LIN {X 0,Y 310.655,Z 525.848,A -85,B 0,C 180,E1 -15761.749,E2 -15761.749} C_VEL
LIN {X 0,Y 310.622,Z 526.997,A -85,B 0,C 180,E1 -15763.368,E2 -15763.368} C_VEL
LIN {X 0,Y 310.6,Z 527.515,A -85,B 0,C 180,E1 -15765.756,E2 -15765.756} C_VEL
LIN {X 0,Y 310.891,Z 526.626,A -85,B 0,C 180,E1 -15768.294,E2 -15768.294} C_VEL
LIN {X 0,Y 311.191,Z 525.391,A -85,B 0,C 180,E1 -15769.802,E2 -15769.802} C_VEL
LIN {X 0,Y 311.807,Z 522.832,A -85,B 0,C 180,E1 -15771.834,E2 -15771.834} C_VEL
LIN {X 0,Y 312.562,Z 519.175,A -85,B 0,C 180,E1 -15773.875,E2 -15773.875} C_VEL
LIN {X 0,Y 313.548,Z 514.547,A -85,B 0,C 180,E1 -15775.824,E2 -15775.824} C_VEL
LIN {X 0,Y 314.939,Z 508.045,A -85,B 0,C 180,E1 -15777.946,E2 -15777.946} C_VEL
LIN {X 0,Y 316.348,Z 501.394,A -85,B 0,C 180,E1 -15779.675,E2 -15779.675} C_VEL
LIN {X 0,Y 317.833,Z 493.733,A -85,B 0,C 180,E1 -15781.308,E2 -15781.308} C_VEL
LIN {X 0,Y 319.671,Z 484.109,A -85,B 0,C 180,E1 -15782.966,E2 -15782.966} C_VEL
LIN {X 0,Y 321.573,Z 473.195,A -85,B 0,C 180,E1 -15784.445,E2 -15784.445} C_VEL
LIN {X 0,Y 323.064,Z 462.681,A -85,B 0,C 180,E1 -15785.587,E2 -15785.587} C_VEL
LIN {X 0,Y 324.486,Z 450.756,A -85,B 0,C 180,E1 -15786.597,E2 -15786.597} C_VEL
LIN {X 0,Y 325.603,Z 438.12,A -85,B 0,C 180,E1 -15787.378,E2 -15787.378} C_VEL
LIN {X 0,Y 326.342,Z 425.507,A -85,B 0,C 180,E1 -15787.912,E2 -15787.912} C_VEL
LIN {X 0,Y 327.507,Z 389.604,A -85,B 0,C 180,E1 -15788.742,E2 -15788.742} C_VEL
LIN {X 0,Y 328.624,Z 348.659,A -85,B 0,C 180,E1 -15789.655,E2 -15789.655} C_VEL
LIN {X 0,Y 322.438,Z 334.155,A -85,B 0,C 180,E1 -15790.674,E2 -15790.674} C_VEL
LIN {X 0,Y 315.363,Z 320.101,A -85,B 0,C 180,E1 -15791.839,E2 -15791.839} C_VEL
LIN {X 0,Y 314.876,Z 319.253,A -85,B 0,C 180,E1 -15791.919,E2 -15791.919} C_VEL
LIN {X 0,Y 313.157,Z 317.364,A -85,B 0,C 180,E1 -15792.239,E2 -15792.239} C_VEL
LIN {X 0,Y 310.38,Z 316.136,A -85,B 0,C 180,E1 -15792.856,E2 -15792.856} C_VEL
LIN {X 0,Y 306.923,Z 314.284,A -85,B 0,C 180,E1 -15793.938,E2 -15793.938} C_VEL
LIN {X 0,Y 305.535,Z 312.708,A -85,B 0,C 180,E1 -15794.807,E2 -15794.807} C_VEL
LIN {X 0,Y 305.384,Z 312.449,A -85,B 0,C 180,E1 -15795.209,E2 -15795.209} C_VEL
LIN {X 0,Y 305.443,Z 312.442,A -85,B 0,C 180,E1 -15798.143,E2 -15798.143} C_VEL
LIN {X 0,Y 305.478,Z 312.425,A -85,B 0,C 180,E1 -15801.598,E2 -15801.598} C_VEL
LIN {X 0,Y 305.464,Z 312.435,A -85,B 0,C 180,E1 -15804.887,E2 -15804.887} C_VEL
LIN {X 0,Y 305.454,Z 312.436,A -85,B 0,C 180,E1 -15808.355,E2 -15808.355} C_VEL
LIN {X 0,Y 305.523,Z 312.427,A -85,B 0,C 180,E1 -15811.114,E2 -15811.114} C_VEL
LIN {X 0,Y 305.573,Z 312.418,A -85,B 0,C 180,E1 -15814.088,E2 -15814.088} C_VEL
LIN {X 0,Y 305.502,Z 312.427,A -85,B 0,C 180,E1 -15818.403,E2 -15818.403} C_VEL
LIN {X 0,Y 305.592,Z 312.409,A -85,B 0,C 180,E1 -15821.218,E2 -15821.218} C_VEL
LIN {X 0,Y 305.65,Z 312.401,A -85,B 0,C 180,E1 -15825.349,E2 -15825.349} C_VEL
LIN {X 0,Y 305.64,Z 312.406,A -85,B 0,C 180,E1 -15829.4,E2 -15829.4} C_VEL
LIN {X 0,Y 305.815,Z 312.388,A -85,B 0,C 180,E1 -15832.074,E2 -15832.074} C_VEL
LIN {X 0,Y 305.688,Z 312.4,A -85,B 0,C 180,E1 -15834.723,E2 -15834.723} C_VEL
LIN {X 0,Y 305.956,Z 312.37,A -85,B 0,C 180,E1 -15838.684,E2 -15838.684} C_VEL
LIN {X 0,Y 305.956,Z 312.357,A -85,B 0,C 180,E1 -15841.316,E2 -15841.316} C_VEL
LIN {X 0,Y 305.852,Z 312.373,A -85,B 0,C 180,E1 -15846.597,E2 -15846.597} C_VEL
LIN {X 0,Y 305.737,Z 312.396,A -85,B 0,C 180,E1 -15849.26,E2 -15849.26} C_VEL
LIN {X 0,Y 305.59,Z 312.416,A -85,B 0,C 180,E1 -15853.296,E2 -15853.296} C_VEL
LIN {X 0,Y 305.595,Z 312.407,A -85,B 0,C 180,E1 -15856.02,E2 -15856.02} C_VEL
LIN {X 0,Y 305.577,Z 312.418,A -85,B 0,C 180,E1 -15859.444,E2 -15859.444} C_VEL
LIN {X 0,Y 305.488,Z 312.434,A -85,B 0,C 180,E1 -15863.039,E2 -15863.039} C_VEL
LIN {X 0,Y 305.528,Z 312.416,A -85,B 0,C 180,E1 -15866.219,E2 -15866.219} C_VEL
LIN {X 0,Y 305.497,Z 312.424,A -85,B 0,C 180,E1 -15869.05,E2 -15869.05} C_VEL
LIN {X 0,Y 305.446,Z 312.436,A -85,B 0,C 180,E1 -15871.952,E2 -15871.952} C_VEL
LIN {X 0,Y 305.464,Z 312.432,A -85,B 0,C 180,E1 -15875.113,E2 -15875.113} C_VEL
LIN {X 0,Y 305.45,Z 312.435,A -85,B 0,C 180,E1 -15878.528,E2 -15878.528} C_VEL
LIN {X 0,Y 305.457,Z 312.437,A -85,B 0,C 180,E1 -15882.586,E2 -15882.586} C_VEL
LIN {X 0,Y 305.427,Z 312.438,A -85,B 0,C 180,E1 -15886.345,E2 -15886.345} C_VEL
LIN {X 0,Y 305.46,Z 312.429,A -85,B 0,C 180,E1 -15889.892,E2 -15889.892} C_VEL
LIN {X 0,Y 305.499,Z 312.616,A -85,B 0,C 180,E1 -15893.627,E2 -15893.627} C_VEL
LIN {X 0,Y 308.251,Z 323.052,A -85,B 0,C 180,E1 -15897.288,E2 -15897.288} C_VEL
LIN {X 0,Y 310.521,Z 332.941,A -85,B 0,C 180,E1 -15900.51,E2 -15900.51} C_VEL
LIN {X 0,Y 311.361,Z 336.906,A -85,B 0,C 180,E1 -15901.679,E2 -15901.679} C_VEL
LIN {X 0,Y 314.684,Z 344.996,A -85,B 0,C 180,E1 -15902.285,E2 -15902.285} C_VEL
LIN {X 0,Y 319.531,Z 367.922,A -85,B 0,C 180,E1 -15903.422,E2 -15903.422} C_VEL
LIN {X 0,Y 321.715,Z 382.032,A -85,B 0,C 180,E1 -15904.015,E2 -15904.015} C_VEL
LIN {X 0,Y 319.792,Z 445.993,A -85,B 0,C 180,E1 -15905.492,E2 -15905.492} C_VEL
LIN {X 0,Y 318.71,Z 459.732,A -85,B 0,C 180,E1 -15906.053,E2 -15906.053} C_VEL
LIN {X 0,Y 317.279,Z 472.616,A -85,B 0,C 180,E1 -15906.847,E2 -15906.847} C_VEL
LIN {X 0,Y 315.482,Z 485.127,A -85,B 0,C 180,E1 -15907.918,E2 -15907.918} C_VEL
LIN {X 0,Y 313.614,Z 496.298,A -85,B 0,C 180,E1 -15909.16,E2 -15909.16} C_VEL
LIN {X 0,Y 311.639,Z 506.4,A -85,B 0,C 180,E1 -15910.57,E2 -15910.57} C_VEL
LIN {X 0,Y 309.74,Z 515.84,A -85,B 0,C 180,E1 -15912.23,E2 -15912.23} C_VEL
LIN {X 0,Y 308.099,Z 524.424,A -85,B 0,C 180,E1 -15914.113,E2 -15914.113} C_VEL
LIN {X 0,Y 306.566,Z 531.627,A -85,B 0,C 180,E1 -15916.071,E2 -15916.071} C_VEL
LIN {X 0,Y 305.309,Z 537.408,A -85,B 0,C 180,E1 -15918.042,E2 -15918.042} C_VEL
LIN {X 0,Y 304.501,Z 541.984,A -85,B 0,C 180,E1 -15920.031,E2 -15920.031} C_VEL
LIN {X 0,Y 303.991,Z 545.486,A -85,B 0,C 180,E1 -15922.026,E2 -15922.026} C_VEL
LIN {X 0,Y 303.66,Z 548.358,A -85,B 0,C 180,E1 -15924.388,E2 -15924.388} C_VEL
LIN {X 0,Y 303.633,Z 549.588,A -85,B 0,C 180,E1 -15926.017,E2 -15926.017} C_VEL
LIN {X 0,Y 303.623,Z 550.172,A -85,B 0,C 180,E1 -15927.346,E2 -15927.346} C_VEL
LIN {X 0,Y 303.607,Z 550.326,A -85,B 0,C 180,E1 -15928.673,E2 -15928.673} C_VEL
LIN {X 0,Y 303.669,Z 550.081,A -85,B 0,C 180,E1 -15929.999,E2 -15929.999} C_VEL
LIN {X 0,Y 303.635,Z 549.443,A -85,B 0,C 180,E1 -15931.325,E2 -15931.325} C_VEL
LIN {X 0,Y 303.645,Z 548.412,A -85,B 0,C 180,E1 -15932.652,E2 -15932.652} C_VEL
LIN {X 0,Y 303.67,Z 546.932,A -85,B 0,C 180,E1 -15933.98,E2 -15933.98} C_VEL
LIN {X 0,Y 303.729,Z 544.305,A -85,B 0,C 180,E1 -15935.743,E2 -15935.743} C_VEL
LIN {X 0,Y 303.938,Z 539.781,A -85,B 0,C 180,E1 -15937.974,E2 -15937.974} C_VEL
LIN {X 0,Y 304.438,Z 533.452,A -85,B 0,C 180,E1 -15940.305,E2 -15940.305} C_VEL
LIN {X 0,Y 305.125,Z 526.543,A -85,B 0,C 180,E1 -15942.3,E2 -15942.3} C_VEL
LIN {X 0,Y 306.006,Z 519.49,A -85,B 0,C 180,E1 -15943.953,E2 -15943.953} C_VEL
LIN {X 0,Y 307.069,Z 510.98,A -85,B 0,C 180,E1 -15945.599,E2 -15945.599} C_VEL
LIN {X 0,Y 308.256,Z 500.429,A -85,B 0,C 180,E1 -15947.24,E2 -15947.24} C_VEL
LIN {X 0,Y 309.191,Z 491.41,A -85,B 0,C 180,E1 -15948.383,E2 -15948.383} C_VEL
LIN {X 0,Y 310.442,Z 480.31,A -85,B 0,C 180,E1 -15949.506,E2 -15949.506} C_VEL
LIN {X 0,Y 311.569,Z 467.989,A -85,B 0,C 180,E1 -15950.463,E2 -15950.463} C_VEL
LIN {X 0,Y 312.495,Z 455.009,A -85,B 0,C 180,E1 -15951.175,E2 -15951.175} C_VEL
LIN {X 0,Y 313.083,Z 441.167,A -85,B 0,C 180,E1 -15951.652,E2 -15951.652} C_VEL
LIN {X 0,Y 314.281,Z 378.975,A -85,B 0,C 180,E1 -15953.068,E2 -15953.068} C_VEL
LIN {X 0,Y 308.693,Z 337.549,A -85,B 0,C 180,E1 -15954.448,E2 -15954.448} C_VEL
LIN {X 0,Y 309.29,Z 331.837,A -85,B 0,C 180,E1 -15955.938,E2 -15955.938} C_VEL
LIN {X 0,Y 307.581,Z 322.176,A -85,B 0,C 180,E1 -15958.673,E2 -15958.673} C_VEL
LIN {X 0,Y 305.465,Z 312.437,A -85,B 0,C 180,E1 -15961.578,E2 -15961.578} C_VEL
LIN {X 0,Y 305.459,Z 312.433,A -85,B 0,C 180,E1 -15965.112,E2 -15965.112} C_VEL
LIN {X 0,Y 305.463,Z 312.435,A -85,B 0,C 180,E1 -15968.532,E2 -15968.532} C_VEL
LIN {X 0,Y 305.45,Z 312.438,A -85,B 0,C 180,E1 -15972.585,E2 -15972.585} C_VEL
LIN {X 0,Y 305.468,Z 312.432,A -85,B 0,C 180,E1 -15977.409,E2 -15977.409} C_VEL
LIN {X 0,Y 305.489,Z 312.428,A -85,B 0,C 180,E1 -15981.599,E2 -15981.599} C_VEL
LIN {X 0,Y 305.457,Z 312.437,A -85,B 0,C 180,E1 -15984.886,E2 -15984.886} C_VEL
LIN {X 0,Y 305.449,Z 312.434,A -85,B 0,C 180,E1 -15988.353,E2 -15988.353} C_VEL
LIN {X 0,Y 305.514,Z 312.429,A -85,B 0,C 180,E1 -15991.113,E2 -15991.113} C_VEL
LIN {X 0,Y 305.564,Z 312.419,A -85,B 0,C 180,E1 -15994.087,E2 -15994.087} C_VEL
LIN {X 0,Y 305.492,Z 312.429,A -85,B 0,C 180,E1 -15998.402,E2 -15998.402} C_VEL
LIN {X 0,Y 305.582,Z 312.418,A -85,B 0,C 180,E1 -16001.217,E2 -16001.217} C_VEL
LIN {X 0,Y 305.641,Z 312.413,A -85,B 0,C 180,E1 -16005.349,E2 -16005.349} C_VEL
LIN {X 0,Y 305.63,Z 312.416,A -85,B 0,C 180,E1 -16009.399,E2 -16009.399} C_VEL
LIN {X 0,Y 305.804,Z 312.386,A -85,B 0,C 180,E1 -16012.074,E2 -16012.074} C_VEL
LIN {X 0,Y 305.68,Z 312.399,A -85,B 0,C 180,E1 -16014.723,E2 -16014.723} C_VEL
LIN {X 0,Y 305.948,Z 312.371,A -85,B 0,C 180,E1 -16018.684,E2 -16018.684} C_VEL
LIN {X 0,Y 305.949,Z 312.373,A -85,B 0,C 180,E1 -16021.316,E2 -16021.316} C_VEL
LIN {X 0,Y 305.666,Z 312.402,A -85,B 0,C 180,E1 -16025.277,E2 -16025.277} C_VEL
LIN {X 0,Y 305.755,Z 312.396,A -85,B 0,C 180,E1 -16027.927,E2 -16027.927} C_VEL
LIN {X 0,Y 305.595,Z 312.42,A -85,B 0,C 180,E1 -16031.946,E2 -16031.946} C_VEL
LIN {X 0,Y 305.63,Z 312.409,A -85,B 0,C 180,E1 -16035.035,E2 -16035.035} C_VEL
LIN {X 0,Y 305.568,Z 312.419,A -85,B 0,C 180,E1 -16039.445,E2 -16039.445} C_VEL
LIN {X 0,Y 305.479,Z 312.43,A -85,B 0,C 180,E1 -16043.04,E2 -16043.04} C_VEL
LIN {X 0,Y 305.54,Z 312.427,A -85,B 0,C 180,E1 -16046.228,E2 -16046.228} C_VEL
LIN {X 0,Y 305.489,Z 312.429,A -85,B 0,C 180,E1 -16049.051,E2 -16049.051} C_VEL
LIN {X 0,Y 305.458,Z 312.43,A -85,B 0,C 180,E1 -16053.518,E2 -16053.518} C_VEL
LIN {X 0,Y 305.463,Z 312.436,A -85,B 0,C 180,E1 -16056.741,E2 -16056.741} C_VEL
LIN {X 0,Y 305.403,Z 312.442,A -85,B 0,C 180,E1 -16060.591,E2 -16060.591} C_VEL
LIN {X 0,Y 305.416,Z 312.436,A -85,B 0,C 180,E1 -16063.657,E2 -16063.657} C_VEL
LIN {X 0,Y 305.431,Z 312.437,A -85,B 0,C 180,E1 -16067.42,E2 -16067.42} C_VEL
LIN {X 0,Y 305.456,Z 312.434,A -85,B 0,C 180,E1 -16071.596,E2 -16071.596} C_VEL
LIN {X 0,Y 305.459,Z 312.436,A -85,B 0,C 180,E1 -16074.888,E2 -16074.888} C_VEL
LIN {X 0,Y 305.439,Z 312.435,A -85,B 0,C 180,E1 -16078.36,E2 -16078.36} C_VEL
LIN {X 0,Y 305.472,Z 312.434,A -85,B 0,C 180,E1 -16081.11,E2 -16081.11} C_VEL
LIN {X 0,Y 305.496,Z 312.429,A -85,B 0,C 180,E1 -16084.083,E2 -16084.083} C_VEL
LIN {X 0,Y 305.472,Z 312.433,A -85,B 0,C 180,E1 -16086.977,E2 -16086.977} C_VEL
LIN {X 0,Y 305.542,Z 312.425,A -85,B 0,C 180,E1 -16091.216,E2 -16091.216} C_VEL
LIN {X 0,Y 305.628,Z 312.415,A -85,B 0,C 180,E1 -16095.349,E2 -16095.349} C_VEL
LIN {X 0,Y 305.627,Z 312.566,A -85,B 0,C 180,E1 -16098.225,E2 -16098.225} C_VEL
LIN {X 0,Y 306.516,Z 316.718,A -85,B 0,C 180,E1 -16099.508,E2 -16099.508} C_VEL
LIN {X 0,Y 312.875,Z 335.486,A -85,B 0,C 180,E1 -16100.394,E2 -16100.394} C_VEL
LIN {X 0,Y 314.978,Z 347.517,A -85,B 0,C 180,E1 -16100.819,E2 -16100.819} C_VEL
LIN {X 0,Y 313.14,Z 424.528,A -85,B 0,C 180,E1 -16102.586,E2 -16102.586} C_VEL
LIN {X 0,Y 312.537,Z 437.514,A -85,B 0,C 180,E1 -16103.14,E2 -16103.14} C_VEL
LIN {X 0,Y 311.726,Z 450.087,A -85,B 0,C 180,E1 -16103.935,E2 -16103.935} C_VEL
LIN {X 0,Y 310.797,Z 461.998,A -85,B 0,C 180,E1 -16104.968,E2 -16104.968} C_VEL
LIN {X 0,Y 309.618,Z 473.529,A -85,B 0,C 180,E1 -16106.259,E2 -16106.259} C_VEL
LIN {X 0,Y 308.386,Z 483.881,A -85,B 0,C 180,E1 -16107.715,E2 -16107.715} C_VEL
LIN {X 0,Y 307.181,Z 493.179,A -85,B 0,C 180,E1 -16109.346,E2 -16109.346} C_VEL
LIN {X 0,Y 306.032,Z 502.185,A -85,B 0,C 180,E1 -16111.317,E2 -16111.317} C_VEL
LIN {X 0,Y 305.201,Z 509.434,A -85,B 0,C 180,E1 -16113.301,E2 -16113.301} C_VEL
LIN {X 0,Y 304.55,Z 515.23,A -85,B 0,C 180,E1 -16115.297,E2 -16115.297} C_VEL
LIN {X 0,Y 304.145,Z 519.658,A -85,B 0,C 180,E1 -16117.236,E2 -16117.236} C_VEL
LIN {X 0,Y 303.766,Z 523.266,A -85,B 0,C 180,E1 -16119.321,E2 -16119.321} C_VEL
LIN {X 0,Y 303.584,Z 524.997,A -85,B 0,C 180,E1 -16120.674,E2 -16120.674} C_VEL
LIN {X 0,Y 303.542,Z 526.313,A -85,B 0,C 180,E1 -16122.028,E2 -16122.028} C_VEL
LIN {X 0,Y 303.531,Z 527.273,A -85,B 0,C 180,E1 -16123.473,E2 -16123.473} C_VEL
LIN {X 0,Y 303.531,Z 527.757,A -85,B 0,C 180,E1 -16126.133,E2 -16126.133} C_VEL
LIN {X 0,Y 303.866,Z 526.883,A -85,B 0,C 180,E1 -16128.508,E2 -16128.508} C_VEL
LIN {X 0,Y 304.21,Z 525.403,A -85,B 0,C 180,E1 -16130.276,E2 -16130.276} C_VEL
LIN {X 0,Y 305.079,Z 521.93,A -85,B 0,C 180,E1 -16132.858,E2 -16132.858} C_VEL
LIN {X 0,Y 306.084,Z 517.421,A -85,B 0,C 180,E1 -16135.137,E2 -16135.137} C_VEL
LIN {X 0,Y 307.33,Z 511.945,A -85,B 0,C 180,E1 -16137.217,E2 -16137.217} C_VEL
LIN {X 0,Y 308.942,Z 504.997,A -85,B 0,C 180,E1 -16139.282,E2 -16139.282} C_VEL
LIN {X 0,Y 310.561,Z 497.418,A -85,B 0,C 180,E1 -16141.088,E2 -16141.088} C_VEL
LIN {X 0,Y 312.218,Z 489.107,A -85,B 0,C 180,E1 -16142.7,E2 -16142.7} C_VEL
LIN {X 0,Y 314.216,Z 478.662,A -85,B 0,C 180,E1 -16144.313,E2 -16144.313} C_VEL
LIN {X 0,Y 316.11,Z 467.254,A -85,B 0,C 180,E1 -16145.705,E2 -16145.705} C_VEL
LIN {X 0,Y 317.626,Z 455.882,A -85,B 0,C 180,E1 -16146.793,E2 -16146.793} C_VEL
LIN {X 0,Y 318.875,Z 444.501,A -85,B 0,C 180,E1 -16147.615,E2 -16147.615} C_VEL
LIN {X 0,Y 319.822,Z 431.965,A -85,B 0,C 180,E1 -16148.274,E2 -16148.274} C_VEL
LIN {X 0,Y 320.387,Z 419.421,A -85,B 0,C 180,E1 -16148.696,E2 -16148.696} C_VEL
LIN {X 0,Y 322.479,Z 350.403,A -85,B 0,C 180,E1 -16150.251,E2 -16150.251} C_VEL
LIN {X 0,Y 315.024,Z 333.6,A -85,B 0,C 180,E1 -16151.517,E2 -16151.517} C_VEL
LIN {X 0,Y 308.345,Z 320.625,A -85,B 0,C 180,E1 -16152.669,E2 -16152.669} C_VEL
LIN {X 0,Y 306.666,Z 317.222,A -85,B 0,C 180,E1 -16153.018,E2 -16153.018} C_VEL
LIN {X 0,Y 305.38,Z 312.451,A -85,B 0,C 180,E1 -16154.77,E2 -16154.77} C_VEL
LIN {X 0,Y 305.384,Z 312.449,A -85,B 0,C 180,E1 -16155.209,E2 -16155.209} C_VEL
LIN {X 0,Y 304.768,Z 312.52,A -85,B 0,C 180,E1 -16156.31,E2 -16156.31} C_VEL
LIN {X 0,Y 301.968,Z 312.875,A -85,B 0,C 180,E1 -16158.104,E2 -16158.104} C_VEL
LIN {X 0,Y 299.556,Z 313.166,A -85,B 0,C 180,E1 -16159.559,E2 -16159.559} C_VEL
LIN {X 0,Y 298.499,Z 313.29,A -85,B 0,C 180,E1 -16160.686,E2 -16160.686} C_VEL
LIN {X 0,Y 298.403,Z 313.302,A -85,B 0,C 180,E1 -16161.068,E2 -16161.068} C_VEL
LIN {X 0,Y 298.421,Z 313.311,A -85,B 0,C 180,E1 -16163.93,E2 -16163.93} C_VEL
LIN {X 0,Y 298.398,Z 313.315,A -85,B 0,C 180,E1 -16167.983,E2 -16167.983} C_VEL
LIN {X 0,Y 298.466,Z 313.306,A -85,B 0,C 180,E1 -16171.904,E2 -16171.904} C_VEL
LIN {X 0,Y 298.488,Z 313.304,A -85,B 0,C 180,E1 -16174.924,E2 -16174.924} C_VEL
LIN {X 0,Y 298.452,Z 313.308,A -85,B 0,C 180,E1 -16179.315,E2 -16179.315} C_VEL
LIN {X 0,Y 298.54,Z 313.293,A -85,B 0,C 180,E1 -16182.179,E2 -16182.179} C_VEL
LIN {X 0,Y 298.595,Z 313.282,A -85,B 0,C 180,E1 -16184.995,E2 -16184.995} C_VEL
LIN {X 0,Y 298.595,Z 313.287,A -85,B 0,C 180,E1 -16189.147,E2 -16189.147} C_VEL
LIN {X 0,Y 298.761,Z 313.264,A -85,B 0,C 180,E1 -16191.886,E2 -16191.886} C_VEL
LIN {X 0,Y 298.66,Z 313.275,A -85,B 0,C 180,E1 -16194.599,E2 -16194.599} C_VEL
LIN {X 0,Y 298.923,Z 313.247,A -85,B 0,C 180,E1 -16198.653,E2 -16198.653} C_VEL
LIN {X 0,Y 298.923,Z 313.233,A -85,B 0,C 180,E1 -16201.347,E2 -16201.347} C_VEL
LIN {X 0,Y 298.798,Z 313.252,A -85,B 0,C 180,E1 -16206.754,E2 -16206.754} C_VEL
LIN {X 0,Y 298.682,Z 313.275,A -85,B 0,C 180,E1 -16209.48,E2 -16209.48} C_VEL
LIN {X 0,Y 298.553,Z 313.292,A -85,B 0,C 180,E1 -16213.615,E2 -16213.615} C_VEL
LIN {X 0,Y 298.55,Z 313.284,A -85,B 0,C 180,E1 -16216.409,E2 -16216.409} C_VEL
LIN {X 0,Y 298.512,Z 313.298,A -85,B 0,C 180,E1 -16219.654,E2 -16219.654} C_VEL
LIN {X 0,Y 298.43,Z 313.31,A -85,B 0,C 180,E1 -16223.6,E2 -16223.6} C_VEL
LIN {X 0,Y 298.487,Z 313.295,A -85,B 0,C 180,E1 -16226.575,E2 -16226.575} C_VEL
LIN {X 0,Y 298.422,Z 313.301,A -85,B 0,C 180,E1 -16229.641,E2 -16229.641} C_VEL
LIN {X 0,Y 298.397,Z 313.312,A -85,B 0,C 180,E1 -16232.8,E2 -16232.8} C_VEL
LIN {X 0,Y 298.448,Z 313.305,A -85,B 0,C 180,E1 -16236.807,E2 -16236.807} C_VEL
LIN {X 0,Y 298.389,Z 313.313,A -85,B 0,C 180,E1 -16241.087,E2 -16241.087} C_VEL
LIN {X 0,Y 298.401,Z 313.313,A -85,B 0,C 180,E1 -16243.103,E2 -16243.103} C_VEL
LIN {X 0,Y 298.405,Z 313.315,A -85,B 0,C 180,E1 -16246.921,E2 -16246.921} C_VEL
LIN {X 0,Y 298.401,Z 313.303,A -85,B 0,C 180,E1 -16251.007,E2 -16251.007} C_VEL
LIN {X 0,Y 298.415,Z 313.327,A -85,B 0,C 180,E1 -16252.777,E2 -16252.777} C_VEL
LIN {X 0,Y 300.934,Z 322.839,A -85,B 0,C 180,E1 -16256.252,E2 -16256.252} C_VEL
LIN {X 0,Y 303.379,Z 333.131,A -85,B 0,C 180,E1 -16259.744,E2 -16259.744} C_VEL
LIN {X 0,Y 304.133,Z 336.54,A -85,B 0,C 180,E1 -16260.785,E2 -16260.785} C_VEL
LIN {X 0,Y 308.933,Z 347.604,A -85,B 0,C 180,E1 -16261.683,E2 -16261.683} C_VEL
LIN {X 0,Y 313.606,Z 370.116,A -85,B 0,C 180,E1 -16262.833,E2 -16262.833} C_VEL
LIN {X 0,Y 315.577,Z 383.159,A -85,B 0,C 180,E1 -16263.394,E2 -16263.394} C_VEL
LIN {X 0,Y 313.642,Z 445.184,A -85,B 0,C 180,E1 -16264.846,E2 -16264.846} C_VEL
LIN {X 0,Y 312.571,Z 458.354,A -85,B 0,C 180,E1 -16265.375,E2 -16265.375} C_VEL
LIN {X 0,Y 311.074,Z 471.572,A -85,B 0,C 180,E1 -16266.181,E2 -16266.181} C_VEL
LIN {X 0,Y 309.419,Z 482.714,A -85,B 0,C 180,E1 -16267.109,E2 -16267.109} C_VEL
LIN {X 0,Y 307.49,Z 494.272,A -85,B 0,C 180,E1 -16268.373,E2 -16268.373} C_VEL
LIN {X 0,Y 305.394,Z 504.704,A -85,B 0,C 180,E1 -16269.806,E2 -16269.806} C_VEL
LIN {X 0,Y 303.365,Z 514.296,A -85,B 0,C 180,E1 -16271.459,E2 -16271.459} C_VEL
LIN {X 0,Y 301.744,Z 522.177,A -85,B 0,C 180,E1 -16273.151,E2 -16273.151} C_VEL
LIN {X 0,Y 300.184,Z 529.466,A -85,B 0,C 180,E1 -16275.075,E2 -16275.075} C_VEL
LIN {X 0,Y 298.735,Z 535.606,A -85,B 0,C 180,E1 -16277.085,E2 -16277.085} C_VEL
LIN {X 0,Y 297.743,Z 540.503,A -85,B 0,C 180,E1 -16279.114,E2 -16279.114} C_VEL
LIN {X 0,Y 297.09,Z 544.302,A -85,B 0,C 180,E1 -16281.154,E2 -16281.154} C_VEL
LIN {X 0,Y 296.691,Z 547.099,A -85,B 0,C 180,E1 -16283.197,E2 -16283.197} C_VEL
LIN {X 0,Y 296.53,Z 549.382,A -85,B 0,C 180,E1 -16285.922,E2 -16285.922} C_VEL
LIN {X 0,Y 296.548,Z 549.932,A -85,B 0,C 180,E1 -16287.282,E2 -16287.282} C_VEL
LIN {X 0,Y 296.581,Z 549.78,A -85,B 0,C 180,E1 -16289.999,E2 -16289.999} C_VEL
LIN {X 0,Y 296.551,Z 549.118,A -85,B 0,C 180,E1 -16291.357,E2 -16291.357} C_VEL
LIN {X 0,Y 296.57,Z 548.057,A -85,B 0,C 180,E1 -16292.716,E2 -16292.716} C_VEL
LIN {X 0,Y 296.586,Z 546.533,A -85,B 0,C 180,E1 -16294.075,E2 -16294.075} C_VEL
LIN {X 0,Y 296.676,Z 543.446,A -85,B 0,C 180,E1 -16296.118,E2 -16296.118} C_VEL
LIN {X 0,Y 296.872,Z 539.273,A -85,B 0,C 180,E1 -16298.165,E2 -16298.165} C_VEL
LIN {X 0,Y 297.407,Z 532.882,A -85,B 0,C 180,E1 -16300.552,E2 -16300.552} C_VEL
LIN {X 0,Y 298.166,Z 525.907,A -85,B 0,C 180,E1 -16302.592,E2 -16302.592} C_VEL
LIN {X 0,Y 299.037,Z 518.772,A -85,B 0,C 180,E1 -16304.285,E2 -16304.285} C_VEL
LIN {X 0,Y 300.147,Z 510.139,A -85,B 0,C 180,E1 -16305.968,E2 -16305.968} C_VEL
LIN {X 0,Y 301.411,Z 499.451,A -85,B 0,C 180,E1 -16307.644,E2 -16307.644} C_VEL
LIN {X 0,Y 302.478,Z 490.294,A -85,B 0,C 180,E1 -16308.806,E2 -16308.806} C_VEL
LIN {X 0,Y 303.704,Z 478.976,A -85,B 0,C 180,E1 -16309.957,E2 -16309.957} C_VEL
LIN {X 0,Y 304.878,Z 466.224,A -85,B 0,C 180,E1 -16310.933,E2 -16310.933} C_VEL
LIN {X 0,Y 305.792,Z 453.46,A -85,B 0,C 180,E1 -16311.618,E2 -16311.618} C_VEL
LIN {X 0,Y 306.351,Z 440.307,A -85,B 0,C 180,E1 -16312.064,E2 -16312.064} C_VEL
LIN {X 0,Y 307.553,Z 379.683,A -85,B 0,C 180,E1 -16313.472,E2 -16313.472} C_VEL
LIN {X 0,Y 301.85,Z 337.321,A -85,B 0,C 180,E1 -16314.912,E2 -16314.912} C_VEL
LIN {X 0,Y 302.266,Z 332.467,A -85,B 0,C 180,E1 -16316.215,E2 -16316.215} C_VEL
LIN {X 0,Y 300.457,Z 322.781,A -85,B 0,C 180,E1 -16319.035,E2 -16319.035} C_VEL
LIN {X 0,Y 298.422,Z 313.316,A -85,B 0,C 180,E1 -16321.953,E2 -16321.953} C_VEL
LIN {X 0,Y 298.415,Z 313.314,A -85,B 0,C 180,E1 -16326.068,E2 -16326.068} C_VEL
LIN {X 0,Y 298.404,Z 313.311,A -85,B 0,C 180,E1 -16329.485,E2 -16329.485} C_VEL
LIN {X 0,Y 298.394,Z 313.313,A -85,B 0,C 180,E1 -16333.102,E2 -16333.102} C_VEL
LIN {X 0,Y 298.397,Z 313.315,A -85,B 0,C 180,E1 -16336.92,E2 -16336.92} C_VEL
LIN {X 0,Y 298.409,Z 313.312,A -85,B 0,C 180,E1 -16341.002,E2 -16341.002} C_VEL
LIN {X 0,Y 298.426,Z 313.309,A -85,B 0,C 180,E1 -16343.931,E2 -16343.931} C_VEL
LIN {X 0,Y 298.392,Z 313.312,A -85,B 0,C 180,E1 -16347.981,E2 -16347.981} C_VEL
LIN {X 0,Y 298.457,Z 313.304,A -85,B 0,C 180,E1 -16351.904,E2 -16351.904} C_VEL
LIN {X 0,Y 298.478,Z 313.307,A -85,B 0,C 180,E1 -16354.923,E2 -16354.923} C_VEL
LIN {X 0,Y 298.442,Z 313.309,A -85,B 0,C 180,E1 -16359.315,E2 -16359.315} C_VEL
LIN {X 0,Y 298.529,Z 313.29,A -85,B 0,C 180,E1 -16362.179,E2 -16362.179} C_VEL
LIN {X 0,Y 298.585,Z 313.288,A -85,B 0,C 180,E1 -16364.994,E2 -16364.994} C_VEL
LIN {X 0,Y 298.586,Z 313.292,A -85,B 0,C 180,E1 -16369.146,E2 -16369.146} C_VEL
LIN {X 0,Y 298.75,Z 313.265,A -85,B 0,C 180,E1 -16371.886,E2 -16371.886} C_VEL
LIN {X 0,Y 298.651,Z 313.273,A -85,B 0,C 180,E1 -16374.599,E2 -16374.599} C_VEL
LIN {X 0,Y 298.915,Z 313.247,A -85,B 0,C 180,E1 -16378.653,E2 -16378.653} C_VEL
LIN {X 0,Y 298.915,Z 313.249,A -85,B 0,C 180,E1 -16381.347,E2 -16381.347} C_VEL
LIN {X 0,Y 298.635,Z 313.278,A -85,B 0,C 180,E1 -16385.402,E2 -16385.402} C_VEL
LIN {X 0,Y 298.704,Z 313.274,A -85,B 0,C 180,E1 -16388.116,E2 -16388.116} C_VEL
LIN {X 0,Y 298.545,Z 313.297,A -85,B 0,C 180,E1 -16392.232,E2 -16392.232} C_VEL
LIN {X 0,Y 298.598,Z 313.285,A -85,B 0,C 180,E1 -16395.21,E2 -16395.21} C_VEL
LIN {X 0,Y 298.531,Z 313.296,A -85,B 0,C 180,E1 -16399.244,E2 -16399.244} C_VEL
LIN {X 0,Y 298.421,Z 313.309,A -85,B 0,C 180,E1 -16403.601,E2 -16403.601} C_VEL
LIN {X 0,Y 298.482,Z 313.304,A -85,B 0,C 180,E1 -16406.575,E2 -16406.575} C_VEL
LIN {X 0,Y 298.414,Z 313.309,A -85,B 0,C 180,E1 -16409.642,E2 -16409.642} C_VEL
LIN {X 0,Y 298.389,Z 313.314,A -85,B 0,C 180,E1 -16412.801,E2 -16412.801} C_VEL
LIN {X 0,Y 298.435,Z 313.311,A -85,B 0,C 180,E1 -16416.807,E2 -16416.807} C_VEL
LIN {X 0,Y 298.342,Z 313.321,A -85,B 0,C 180,E1 -16421.08,E2 -16421.08} C_VEL
LIN {X 0,Y 298.349,Z 313.322,A -85,B 0,C 180,E1 -16425.036,E2 -16425.036} C_VEL
LIN {X 0,Y 298.344,Z 313.322,A -85,B 0,C 180,E1 -16428.922,E2 -16428.922} C_VEL
LIN {X 0,Y 298.438,Z 313.311,A -85,B 0,C 180,E1 -16433.195,E2 -16433.195} C_VEL
LIN {X 0,Y 298.39,Z 313.317,A -85,B 0,C 180,E1 -16437.201,E2 -16437.201} C_VEL
LIN {X 0,Y 298.399,Z 313.312,A -85,B 0,C 180,E1 -16440.627,E2 -16440.627} C_VEL
LIN {X 0,Y 298.437,Z 313.309,A -85,B 0,C 180,E1 -16444.921,E2 -16444.921} C_VEL
LIN {X 0,Y 298.401,Z 313.312,A -85,B 0,C 180,E1 -16447.864,E2 -16447.864} C_VEL
LIN {X 0,Y 298.503,Z 313.3,A -85,B 0,C 180,E1 -16450.756,E2 -16450.756} C_VEL
LIN {X 0,Y 298.586,Z 313.29,A -85,B 0,C 180,E1 -16454.996,E2 -16454.996} C_VEL
LIN {X 0,Y 298.548,Z 313.366,A -85,B 0,C 180,E1 -16457.856,E2 -16457.856} C_VEL
LIN {X 0,Y 299.361,Z 317.09,A -85,B 0,C 180,E1 -16459.01,E2 -16459.01} C_VEL
LIN {X 0,Y 306.264,Z 337.066,A -85,B 0,C 180,E1 -16459.994,E2 -16459.994} C_VEL
LIN {X 0,Y 308.259,Z 348.823,A -85,B 0,C 180,E1 -16460.416,E2 -16460.416} C_VEL
LIN {X 0,Y 306.394,Z 424.197,A -85,B 0,C 180,E1 -16462.173,E2 -16462.173} C_VEL
LIN {X 0,Y 305.775,Z 437.378,A -85,B 0,C 180,E1 -16462.739,E2 -16462.739} C_VEL
LIN {X 0,Y 304.931,Z 450.06,A -85,B 0,C 180,E1 -16463.55,E2 -16463.55} C_VEL
LIN {X 0,Y 304.028,Z 461.333,A -85,B 0,C 180,E1 -16464.529,E2 -16464.529} C_VEL
LIN {X 0,Y 302.794,Z 473.154,A -85,B 0,C 180,E1 -16465.863,E2 -16465.863} C_VEL
LIN {X 0,Y 301.579,Z 483.465,A -85,B 0,C 180,E1 -16467.33,E2 -16467.33} C_VEL
LIN {X 0,Y 300.28,Z 492.929,A -85,B 0,C 180,E1 -16468.995,E2 -16468.995} C_VEL
LIN {X 0,Y 299.107,Z 502.018,A -85,B 0,C 180,E1 -16471.011,E2 -16471.011} C_VEL
LIN {X 0,Y 298.204,Z 509.346,A -85,B 0,C 180,E1 -16473.041,E2 -16473.041} C_VEL
LIN {X 0,Y 297.576,Z 514.316,A -85,B 0,C 180,E1 -16474.742,E2 -16474.742} C_VEL
LIN {X 0,Y 297.151,Z 519.129,A -85,B 0,C 180,E1 -16476.792,E2 -16476.792} C_VEL
LIN {X 0,Y 296.754,Z 522.838,A -85,B 0,C 180,E1 -16478.856,E2 -16478.856} C_VEL
LIN {X 0,Y 296.475,Z 525.519,A -85,B 0,C 180,E1 -16480.933,E2 -16480.933} C_VEL
LIN {X 0,Y 296.431,Z 526.78,A -85,B 0,C 180,E1 -16482.321,E2 -16482.321} C_VEL
LIN {X 0,Y 296.436,Z 527.599,A -85,B 0,C 180,E1 -16483.715,E2 -16483.715} C_VEL
LIN {X 0,Y 296.385,Z 528,A -85,B 0,C 180,E1 -16485.12,E2 -16485.12} C_VEL
LIN {X 0,Y 296.467,Z 528,A -85,B 0,C 180,E1 -16486.528,E2 -16486.528} C_VEL
LIN {X 0,Y 296.834,Z 527.145,A -85,B 0,C 180,E1 -16488.725,E2 -16488.725} C_VEL
LIN {X 0,Y 297.276,Z 525.415,A -85,B 0,C 180,E1 -16490.771,E2 -16490.771} C_VEL
LIN {X 0,Y 298.091,Z 522.235,A -85,B 0,C 180,E1 -16493.147,E2 -16493.147} C_VEL
LIN {X 0,Y 298.944,Z 518.696,A -85,B 0,C 180,E1 -16495.036,E2 -16495.036} C_VEL
LIN {X 0,Y 300.39,Z 512.781,A -85,B 0,C 180,E1 -16497.438,E2 -16497.438} C_VEL
LIN {X 0,Y 302.122,Z 505.68,A -85,B 0,C 180,E1 -16499.626,E2 -16499.626} C_VEL
LIN {X 0,Y 304.043,Z 497.043,A -85,B 0,C 180,E1 -16501.728,E2 -16501.728} C_VEL
LIN {X 0,Y 305.959,Z 488.023,A -85,B 0,C 180,E1 -16503.456,E2 -16503.456} C_VEL
LIN {X 0,Y 307.944,Z 478.037,A -85,B 0,C 180,E1 -16504.989,E2 -16504.989} C_VEL
LIN {X 0,Y 309.824,Z 467.001,A -85,B 0,C 180,E1 -16506.343,E2 -16506.343} C_VEL
LIN {X 0,Y 311.395,Z 455.506,A -85,B 0,C 180,E1 -16507.443,E2 -16507.443} C_VEL
LIN {X 0,Y 312.789,Z 442.773,A -85,B 0,C 180,E1 -16508.351,E2 -16508.351} C_VEL
LIN {X 0,Y 313.791,Z 429.472,A -85,B 0,C 180,E1 -16509.014,E2 -16509.014} C_VEL
LIN {X 0,Y 314.355,Z 415.85,A -85,B 0,C 180,E1 -16509.413,E2 -16509.413} C_VEL
LIN {X 0,Y 316.488,Z 352.797,A -85,B 0,C 180,E1 -16510.84,E2 -16510.84} C_VEL
LIN {X 0,Y 309.917,Z 337.79,A -85,B 0,C 180,E1 -16512.004,E2 -16512.004} C_VEL
LIN {X 0,Y 303.083,Z 324.392,A -85,B 0,C 180,E1 -16513.227,E2 -16513.227} C_VEL
LIN {X 0,Y 299.484,Z 317.572,A -85,B 0,C 180,E1 -16513.934,E2 -16513.934} C_VEL
LIN {X 0,Y 298.371,Z 313.317,A -85,B 0,C 180,E1 -16515.631,E2 -16515.631} C_VEL
LIN {X 0,Y 298.39,Z 313.321,A -85,B 0,C 180,E1 -16518.912,E2 -16518.912} C_VEL
LIN {X 0,Y 298.403,Z 313.302,A -85,B 0,C 180,E1 -16521.068,E2 -16521.068} C_VEL
LIN {X 0,Y 297.706,Z 313.4,A -85,B 0,C 180,E1 -16522.195,E2 -16522.195} C_VEL
LIN {X 0,Y 294.837,Z 313.757,A -85,B 0,C 180,E1 -16524.031,E2 -16524.031} C_VEL
LIN {X 0,Y 292.427,Z 314.061,A -85,B 0,C 180,E1 -16525.52,E2 -16525.52} C_VEL
LIN {X 0,Y 291.406,Z 314.183,A -85,B 0,C 180,E1 -16526.674,E2 -16526.674} C_VEL
LIN {X 0,Y 291.328,Z 314.192,A -85,B 0,C 180,E1 -16527.065,E2 -16527.065} C_VEL
LIN {X 0,Y 291.385,Z 314.189,A -85,B 0,C 180,E1 -16531.158,E2 -16531.158} C_VEL
LIN {X 0,Y 291.419,Z 314.182,A -85,B 0,C 180,E1 -16534.272,E2 -16534.272} C_VEL
LIN {X 0,Y 291.384,Z 314.181,A -85,B 0,C 180,E1 -16537.3,E2 -16537.3} C_VEL
LIN {X 0,Y 291.46,Z 314.173,A -85,B 0,C 180,E1 -16540.27,E2 -16540.27} C_VEL
LIN {X 0,Y 291.557,Z 314.162,A -85,B 0,C 180,E1 -16544.624,E2 -16544.624} C_VEL
LIN {X 0,Y 291.539,Z 314.168,A -85,B 0,C 180,E1 -16548.881,E2 -16548.881} C_VEL
LIN {X 0,Y 291.711,Z 314.139,A -85,B 0,C 180,E1 -16551.688,E2 -16551.688} C_VEL
LIN {X 0,Y 291.631,Z 314.151,A -85,B 0,C 180,E1 -16554.468,E2 -16554.468} C_VEL
LIN {X 0,Y 291.889,Z 314.123,A -85,B 0,C 180,E1 -16558.62,E2 -16558.62} C_VEL
LIN {X 0,Y 291.889,Z 314.109,A -85,B 0,C 180,E1 -16561.38,E2 -16561.38} C_VEL
LIN {X 0,Y 291.747,Z 314.131,A -85,B 0,C 180,E1 -16566.918,E2 -16566.918} C_VEL
LIN {X 0,Y 291.631,Z 314.154,A -85,B 0,C 180,E1 -16569.712,E2 -16569.712} C_VEL
LIN {X 0,Y 291.523,Z 314.17,A -85,B 0,C 180,E1 -16573.95,E2 -16573.95} C_VEL
LIN {X 0,Y 291.489,Z 314.164,A -85,B 0,C 180,E1 -16576.818,E2 -16576.818} C_VEL
LIN {X 0,Y 291.453,Z 314.177,A -85,B 0,C 180,E1 -16579.875,E2 -16579.875} C_VEL
LIN {X 0,Y 291.384,Z 314.189,A -85,B 0,C 180,E1 -16584.207,E2 -16584.207} C_VEL
LIN {X 0,Y 291.422,Z 314.184,A -85,B 0,C 180,E1 -16587.272,E2 -16587.272} C_VEL
LIN {X 0,Y 291.339,Z 314.183,A -85,B 0,C 180,E1 -16590.437,E2 -16590.437} C_VEL
LIN {X 0,Y 291.346,Z 314.183,A -85,B 0,C 180,E1 -16593.698,E2 -16593.698} C_VEL
LIN {X 0,Y 291.378,Z 314.183,A -85,B 0,C 180,E1 -16597.254,E2 -16597.254} C_VEL
LIN {X 0,Y 291.335,Z 314.19,A -85,B 0,C 180,E1 -16600.642,E2 -16600.642} C_VEL
LIN {X 0,Y 291.292,Z 314.201,A -85,B 0,C 180,E1 -16604.402,E2 -16604.402} C_VEL
LIN {X 0,Y 291.329,Z 314.194,A -85,B 0,C 180,E1 -16608.404,E2 -16608.404} C_VEL
LIN {X 0,Y 291.377,Z 314.276,A -85,B 0,C 180,E1 -16611.964,E2 -16611.964} C_VEL
LIN {X 0,Y 293.804,Z 323.254,A -85,B 0,C 180,E1 -16615.381,E2 -16615.381} C_VEL
LIN {X 0,Y 296.094,Z 332.64,A -85,B 0,C 180,E1 -16618.703,E2 -16618.703} C_VEL
LIN {X 0,Y 296.872,Z 336.135,A -85,B 0,C 180,E1 -16619.832,E2 -16619.832} C_VEL
LIN {X 0,Y 303.239,Z 350.231,A -85,B 0,C 180,E1 -16621.06,E2 -16621.06} C_VEL
LIN {X 0,Y 307.738,Z 372.415,A -85,B 0,C 180,E1 -16622.221,E2 -16622.221} C_VEL
LIN {X 0,Y 309.502,Z 384.018,A -85,B 0,C 180,E1 -16622.741,E2 -16622.741} C_VEL
LIN {X 0,Y 307.459,Z 445.507,A -85,B 0,C 180,E1 -16624.212,E2 -16624.212} C_VEL
LIN {X 0,Y 306.288,Z 459.23,A -85,B 0,C 180,E1 -16624.79,E2 -16624.79} C_VEL
LIN {X 0,Y 304.797,Z 471.586,A -85,B 0,C 180,E1 -16625.568,E2 -16625.568} C_VEL
LIN {X 0,Y 302.934,Z 483.437,A -85,B 0,C 180,E1 -16626.59,E2 -16626.59} C_VEL
LIN {X 0,Y 300.929,Z 494.815,A -85,B 0,C 180,E1 -16627.877,E2 -16627.877} C_VEL
LIN {X 0,Y 298.762,Z 505.108,A -85,B 0,C 180,E1 -16629.337,E2 -16629.337} C_VEL
LIN {X 0,Y 296.691,Z 514.382,A -85,B 0,C 180,E1 -16630.991,E2 -16630.991} C_VEL
LIN {X 0,Y 294.875,Z 522.565,A -85,B 0,C 180,E1 -16632.807,E2 -16632.807} C_VEL
LIN {X 0,Y 293.334,Z 529.551,A -85,B 0,C 180,E1 -16634.718,E2 -16634.718} C_VEL
LIN {X 0,Y 291.787,Z 535.625,A -85,B 0,C 180,E1 -16636.772,E2 -16636.772} C_VEL
LIN {X 0,Y 290.76,Z 540.461,A -85,B 0,C 180,E1 -16638.85,E2 -16638.85} C_VEL
LIN {X 0,Y 290.054,Z 544.201,A -85,B 0,C 180,E1 -16640.938,E2 -16640.938} C_VEL
LIN {X 0,Y 289.609,Z 546.944,A -85,B 0,C 180,E1 -16643.03,E2 -16643.03} C_VEL
LIN {X 0,Y 289.432,Z 549.176,A -85,B 0,C 180,E1 -16645.822,E2 -16645.822} C_VEL
LIN {X 0,Y 289.473,Z 549.681,A -85,B 0,C 180,E1 -16647.216,E2 -16647.216} C_VEL
LIN {X 0,Y 289.496,Z 549.479,A -85,B 0,C 180,E1 -16649.999,E2 -16649.999} C_VEL
LIN {X 0,Y 289.47,Z 548.794,A -85,B 0,C 180,E1 -16651.39,E2 -16651.39} C_VEL
LIN {X 0,Y 289.497,Z 547.69,A -85,B 0,C 180,E1 -16652.782,E2 -16652.782} C_VEL
LIN {X 0,Y 289.485,Z 546.133,A -85,B 0,C 180,E1 -16654.176,E2 -16654.176} C_VEL
LIN {X 0,Y 289.601,Z 542.993,A -85,B 0,C 180,E1 -16656.268,E2 -16656.268} C_VEL
LIN {X 0,Y 289.827,Z 538.765,A -85,B 0,C 180,E1 -16658.365,E2 -16658.365} C_VEL
LIN {X 0,Y 290.384,Z 532.311,A -85,B 0,C 180,E1 -16660.81,E2 -16660.81} C_VEL
LIN {X 0,Y 291.216,Z 525.254,A -85,B 0,C 180,E1 -16662.898,E2 -16662.898} C_VEL
LIN {X 0,Y 292.357,Z 516.388,A -85,B 0,C 180,E1 -16664.975,E2 -16664.975} C_VEL
LIN {X 0,Y 293.543,Z 507.11,A -85,B 0,C 180,E1 -16666.728,E2 -16666.728} C_VEL
LIN {X 0,Y 294.717,Z 497.256,A -85,B 0,C 180,E1 -16668.238,E2 -16668.238} C_VEL
LIN {X 0,Y 295.894,Z 487.688,A -85,B 0,C 180,E1 -16669.421,E2 -16669.421} C_VEL
LIN {X 0,Y 297.205,Z 475.61,A -85,B 0,C 180,E1 -16670.593,E2 -16670.593} C_VEL
LIN {X 0,Y 298.321,Z 463.01,A -85,B 0,C 180,E1 -16671.507,E2 -16671.507} C_VEL
LIN {X 0,Y 299.212,Z 449.861,A -85,B 0,C 180,E1 -16672.162,E2 -16672.162} C_VEL
LIN {X 0,Y 299.755,Z 434.388,A -85,B 0,C 180,E1 -16672.607,E2 -16672.607} C_VEL
LIN {X 0,Y 300.728,Z 379.747,A -85,B 0,C 180,E1 -16673.911,E2 -16673.911} C_VEL
LIN {X 0,Y 295.198,Z 338.581,A -85,B 0,C 180,E1 -16675.34,E2 -16675.34} C_VEL
LIN {X 0,Y 295.033,Z 336.938,A -85,B 0,C 180,E1 -16675.436,E2 -16675.436} C_VEL
LIN {X 0,Y 295.193,Z 333.073,A -85,B 0,C 180,E1 -16676.512,E2 -16676.512} C_VEL
LIN {X 0,Y 293.364,Z 323.376,A -85,B 0,C 180,E1 -16679.412,E2 -16679.412} C_VEL
LIN {X 0,Y 291.348,Z 314.196,A -85,B 0,C 180,E1 -16682.28,E2 -16682.28} C_VEL
LIN {X 0,Y 291.358,Z 314.19,A -85,B 0,C 180,E1 -16685.373,E2 -16685.373} C_VEL
LIN {X 0,Y 291.359,Z 314.189,A -85,B 0,C 180,E1 -16688.839,E2 -16688.839} C_VEL
LIN {X 0,Y 291.315,Z 314.198,A -85,B 0,C 180,E1 -16692.491,E2 -16692.491} C_VEL
LIN {X 0,Y 291.304,Z 314.2,A -85,B 0,C 180,E1 -16696.365,E2 -16696.365} C_VEL
LIN {X 0,Y 291.381,Z 314.188,A -85,B 0,C 180,E1 -16700.516,E2 -16700.516} C_VEL
LIN {X 0,Y 291.419,Z 314.185,A -85,B 0,C 180,E1 -16702.921,E2 -16702.921} C_VEL
LIN {X 0,Y 291.339,Z 314.193,A -85,B 0,C 180,E1 -16706.301,E2 -16706.301} C_VEL
LIN {X 0,Y 291.381,Z 314.187,A -85,B 0,C 180,E1 -16710.259,E2 -16710.259} C_VEL
LIN {X 0,Y 291.409,Z 314.183,A -85,B 0,C 180,E1 -16714.271,E2 -16714.271} C_VEL
LIN {X 0,Y 291.374,Z 314.191,A -85,B 0,C 180,E1 -16717.299,E2 -16717.299} C_VEL
LIN {X 0,Y 291.45,Z 314.176,A -85,B 0,C 180,E1 -16720.27,E2 -16720.27} C_VEL
LIN {X 0,Y 291.532,Z 314.163,A -85,B 0,C 180,E1 -16724.634,E2 -16724.634} C_VEL
LIN {X 0,Y 291.529,Z 314.169,A -85,B 0,C 180,E1 -16728.88,E2 -16728.88} C_VEL
LIN {X 0,Y 291.7,Z 314.144,A -85,B 0,C 180,E1 -16731.688,E2 -16731.688} C_VEL
LIN {X 0,Y 291.622,Z 314.148,A -85,B 0,C 180,E1 -16734.468,E2 -16734.468} C_VEL
LIN {X 0,Y 291.881,Z 314.123,A -85,B 0,C 180,E1 -16738.62,E2 -16738.62} C_VEL
LIN {X 0,Y 291.881,Z 314.126,A -85,B 0,C 180,E1 -16741.38,E2 -16741.38} C_VEL
LIN {X 0,Y 291.65,Z 314.143,A -85,B 0,C 180,E1 -16746.553,E2 -16746.553} C_VEL
LIN {X 0,Y 291.564,Z 314.163,A -85,B 0,C 180,E1 -16749.714,E2 -16749.714} C_VEL
LIN {X 0,Y 291.514,Z 314.174,A -85,B 0,C 180,E1 -16753.951,E2 -16753.951} C_VEL
LIN {X 0,Y 291.479,Z 314.174,A -85,B 0,C 180,E1 -16756.818,E2 -16756.818} C_VEL
LIN {X 0,Y 291.443,Z 314.181,A -85,B 0,C 180,E1 -16759.876,E2 -16759.876} C_VEL
LIN {X 0,Y 291.376,Z 314.191,A -85,B 0,C 180,E1 -16764.208,E2 -16764.208} C_VEL
LIN {X 0,Y 291.416,Z 314.18,A -85,B 0,C 180,E1 -16767.272,E2 -16767.272} C_VEL
LIN {X 0,Y 291.331,Z 314.197,A -85,B 0,C 180,E1 -16770.438,E2 -16770.438} C_VEL
LIN {X 0,Y 291.338,Z 314.189,A -85,B 0,C 180,E1 -16773.699,E2 -16773.699} C_VEL
LIN {X 0,Y 291.362,Z 314.188,A -85,B 0,C 180,E1 -16777.253,E2 -16777.253} C_VEL
LIN {X 0,Y 291.294,Z 314.2,A -85,B 0,C 180,E1 -16780.649,E2 -16780.649} C_VEL
LIN {X 0,Y 291.276,Z 314.199,A -85,B 0,C 180,E1 -16784.405,E2 -16784.405} C_VEL
LIN {X 0,Y 291.291,Z 314.198,A -85,B 0,C 180,E1 -16788.413,E2 -16788.413} C_VEL
LIN {X 0,Y 291.331,Z 314.197,A -85,B 0,C 180,E1 -16791.157,E2 -16791.157} C_VEL
LIN {X 0,Y 291.352,Z 314.191,A -85,B 0,C 180,E1 -16794.627,E2 -16794.627} C_VEL
LIN {X 0,Y 291.363,Z 314.189,A -85,B 0,C 180,E1 -16797.951,E2 -16797.951} C_VEL
LIN {X 0,Y 291.341,Z 314.194,A -85,B 0,C 180,E1 -16801.155,E2 -16801.155} C_VEL
LIN {X 0,Y 291.356,Z 314.19,A -85,B 0,C 180,E1 -16804.268,E2 -16804.268} C_VEL
LIN {X 0,Y 291.363,Z 314.193,A -85,B 0,C 180,E1 -16807.299,E2 -16807.299} C_VEL
LIN {X 0,Y 291.439,Z 314.18,A -85,B 0,C 180,E1 -16810.27,E2 -16810.27} C_VEL
LIN {X 0,Y 291.515,Z 314.171,A -85,B 0,C 180,E1 -16814.654,E2 -16814.654} C_VEL
LIN {X 0,Y 291.512,Z 314.277,A -85,B 0,C 180,E1 -16817.514,E2 -16817.514} C_VEL
LIN {X 0,Y 292.152,Z 317.188,A -85,B 0,C 180,E1 -16818.474,E2 -16818.474} C_VEL
LIN {X 0,Y 299.256,Z 337.364,A -85,B 0,C 180,E1 -16819.517,E2 -16819.517} C_VEL
LIN {X 0,Y 301.348,Z 347.243,A -85,B 0,C 180,E1 -16819.912,E2 -16819.912} C_VEL
LIN {X 0,Y 301.473,Z 353.639,A -85,B 0,C 180,E1 -16820.082,E2 -16820.082} C_VEL
LIN {X 0,Y 299.59,Z 425.02,A -85,B 0,C 180,E1 -16821.787,E2 -16821.787} C_VEL
LIN {X 0,Y 298.947,Z 438.663,A -85,B 0,C 180,E1 -16822.402,E2 -16822.402} C_VEL
LIN {X 0,Y 298.062,Z 451.073,A -85,B 0,C 180,E1 -16823.23,E2 -16823.23} C_VEL
LIN {X 0,Y 297.141,Z 462.132,A -85,B 0,C 180,E1 -16824.232,E2 -16824.232} C_VEL
LIN {X 0,Y 295.906,Z 473.572,A -85,B 0,C 180,E1 -16825.559,E2 -16825.559} C_VEL
LIN {X 0,Y 294.605,Z 484.097,A -85,B 0,C 180,E1 -16827.095,E2 -16827.095} C_VEL
LIN {X 0,Y 293.413,Z 492.624,A -85,B 0,C 180,E1 -16828.629,E2 -16828.629} C_VEL
LIN {X 0,Y 292.168,Z 501.838,A -85,B 0,C 180,E1 -16830.69,E2 -16830.69} C_VEL
LIN {X 0,Y 291.208,Z 509.247,A -85,B 0,C 180,E1 -16832.768,E2 -16832.768} C_VEL
LIN {X 0,Y 290.461,Z 515.196,A -85,B 0,C 180,E1 -16834.859,E2 -16834.859} C_VEL
LIN {X 0,Y 290.029,Z 519.883,A -85,B 0,C 180,E1 -16836.96,E2 -16836.96} C_VEL
LIN {X 0,Y 289.62,Z 523.473,A -85,B 0,C 180,E1 -16839.076,E2 -16839.076} C_VEL
LIN {X 0,Y 289.376,Z 526.037,A -85,B 0,C 180,E1 -16841.204,E2 -16841.204} C_VEL
LIN {X 0,Y 289.354,Z 527.824,A -85,B 0,C 180,E1 -16843.7,E2 -16843.7} C_VEL
LIN {X 0,Y 289.306,Z 528.299,A -85,B 0,C 180,E1 -16845.5,E2 -16845.5} C_VEL
LIN {X 0,Y 289.424,Z 528.242,A -85,B 0,C 180,E1 -16846.942,E2 -16846.942} C_VEL
LIN {X 0,Y 289.786,Z 527.417,A -85,B 0,C 180,E1 -16848.942,E2 -16848.942} C_VEL
LIN {X 0,Y 290.336,Z 525.433,A -85,B 0,C 180,E1 -16851.291,E2 -16851.291} C_VEL
LIN {X 0,Y 291.159,Z 522.51,A -85,B 0,C 180,E1 -16853.473,E2 -16853.473} C_VEL
LIN {X 0,Y 292.198,Z 518.468,A -85,B 0,C 180,E1 -16855.655,E2 -16855.655} C_VEL
LIN {X 0,Y 293.664,Z 512.713,A -85,B 0,C 180,E1 -16857.983,E2 -16857.983} C_VEL
LIN {X 0,Y 295.331,Z 506.364,A -85,B 0,C 180,E1 -16859.983,E2 -16859.983} C_VEL
LIN {X 0,Y 297.254,Z 498.131,A -85,B 0,C 180,E1 -16862.059,E2 -16862.059} C_VEL
LIN {X 0,Y 299.312,Z 488.952,A -85,B 0,C 180,E1 -16863.895,E2 -16863.895} C_VEL
LIN {X 0,Y 301.329,Z 479.357,A -85,B 0,C 180,E1 -16865.421,E2 -16865.421} C_VEL
LIN {X 0,Y 303.345,Z 468.25,A -85,B 0,C 180,E1 -16866.833,E2 -16866.833} C_VEL
LIN {X 0,Y 304.848,Z 458.048,A -85,B 0,C 180,E1 -16867.866,E2 -16867.866} C_VEL
LIN {X 0,Y 306.315,Z 446.163,A -85,B 0,C 180,E1 -16868.793,E2 -16868.793} C_VEL
LIN {X 0,Y 307.383,Z 433.833,A -85,B 0,C 180,E1 -16869.483,E2 -16869.483} C_VEL
LIN {X 0,Y 308.027,Z 422.193,A -85,B 0,C 180,E1 -16869.915,E2 -16869.915} C_VEL
LIN {X 0,Y 310.37,Z 354.501,A -85,B 0,C 180,E1 -16871.495,E2 -16871.495} C_VEL
LIN {X 0,Y 302.698,Z 337.439,A -85,B 0,C 180,E1 -16872.905,E2 -16872.905} C_VEL
LIN {X 0,Y 294.181,Z 321.563,A -85,B 0,C 180,E1 -16874.498,E2 -16874.498} C_VEL
LIN {X 0,Y 292.288,Z 317.886,A -85,B 0,C 180,E1 -16874.927,E2 -16874.927} C_VEL
LIN {X 0,Y 291.335,Z 314.188,A -85,B 0,C 180,E1 -16876.473,E2 -16876.473} C_VEL
LIN {X 0,Y 291.384,Z 314.176,A -85,B 0,C 180,E1 -16880.518,E2 -16880.518} C_VEL
LIN {X 0,Y 291.41,Z 314.191,A -85,B 0,C 180,E1 -16882.92,E2 -16882.92} C_VEL
LIN {X 0,Y 291.328,Z 314.192,A -85,B 0,C 180,E1 -16887.065,E2 -16887.065} C_VEL
LIN {X 0,Y 290.689,Z 314.277,A -85,B 0,C 180,E1 -16888.218,E2 -16888.218} C_VEL
LIN {X 0,Y 287.894,Z 314.621,A -85,B 0,C 180,E1 -16890.099,E2 -16890.099} C_VEL
LIN {X 0,Y 285.507,Z 314.921,A -85,B 0,C 180,E1 -16891.624,E2 -16891.624} C_VEL
LIN {X 0,Y 284.473,Z 315.044,A -85,B 0,C 180,E1 -16892.806,E2 -16892.806} C_VEL
LIN {X 0,Y 284.384,Z 315.054,A -85,B 0,C 180,E1 -16893.206,E2 -16893.206} C_VEL
LIN {X 0,Y 284.368,Z 315.054,A -85,B 0,C 180,E1 -16896.707,E2 -16896.707} C_VEL
LIN {X 0,Y 284.405,Z 315.047,A -85,B 0,C 180,E1 -16901.262,E2 -16901.262} C_VEL
LIN {X 0,Y 284.494,Z 315.042,A -85,B 0,C 180,E1 -16904.459,E2 -16904.459} C_VEL
LIN {X 0,Y 284.49,Z 315.046,A -85,B 0,C 180,E1 -16908.601,E2 -16908.601} C_VEL
LIN {X 0,Y 284.661,Z 315.015,A -85,B 0,C 180,E1 -16911.481,E2 -16911.481} C_VEL
LIN {X 0,Y 284.601,Z 315.027,A -85,B 0,C 180,E1 -16914.331,E2 -16914.331} C_VEL
LIN {X 0,Y 284.856,Z 314.999,A -85,B 0,C 180,E1 -16918.586,E2 -16918.586} C_VEL
LIN {X 0,Y 284.856,Z 314.985,A -85,B 0,C 180,E1 -16921.414,E2 -16921.414} C_VEL
LIN {X 0,Y 284.7,Z 315.01,A -85,B 0,C 180,E1 -16927.09,E2 -16927.09} C_VEL
LIN {X 0,Y 284.568,Z 315.029,A -85,B 0,C 180,E1 -16929.955,E2 -16929.955} C_VEL
LIN {X 0,Y 284.483,Z 315.047,A -85,B 0,C 180,E1 -16934.303,E2 -16934.303} C_VEL
LIN {X 0,Y 284.427,Z 315.047,A -85,B 0,C 180,E1 -16937.248,E2 -16937.248} C_VEL
LIN {X 0,Y 284.379,Z 315.053,A -85,B 0,C 180,E1 -16940.242,E2 -16940.242} C_VEL
LIN {X 0,Y 284.338,Z 315.058,A -85,B 0,C 180,E1 -16944.847,E2 -16944.847} C_VEL
LIN {X 0,Y 284.333,Z 315.066,A -85,B 0,C 180,E1 -16948.011,E2 -16948.011} C_VEL
LIN {X 0,Y 284.298,Z 315.068,A -85,B 0,C 180,E1 -16951.274,E2 -16951.274} C_VEL
LIN {X 0,Y 284.343,Z 315.066,A -85,B 0,C 180,E1 -16955.348,E2 -16955.348} C_VEL
LIN {X 0,Y 284.314,Z 315.066,A -85,B 0,C 180,E1 -16958.169,E2 -16958.169} C_VEL
LIN {X 0,Y 284.271,Z 315.076,A -85,B 0,C 180,E1 -16962.124,E2 -16962.124} C_VEL
LIN {X 0,Y 284.257,Z 315.074,A -85,B 0,C 180,E1 -16966.189,E2 -16966.189} C_VEL
LIN {X 0,Y 284.309,Z 315.062,A -85,B 0,C 180,E1 -16970.024,E2 -16970.024} C_VEL
LIN {X 0,Y 284.357,Z 315.266,A -85,B 0,C 180,E1 -16971.116,E2 -16971.116} C_VEL
LIN {X 0,Y 286.944,Z 324.75,A -85,B 0,C 180,E1 -16974.862,E2 -16974.862} C_VEL
LIN {X 0,Y 289.531,Z 335.537,A -85,B 0,C 180,E1 -16978.779,E2 -16978.779} C_VEL
LIN {X 0,Y 297.286,Z 352.187,A -85,B 0,C 180,E1 -16980.355,E2 -16980.355} C_VEL
LIN {X 0,Y 299.469,Z 361.81,A -85,B 0,C 180,E1 -16980.914,E2 -16980.914} C_VEL
LIN {X 0,Y 302.75,Z 379.894,A -85,B 0,C 180,E1 -16981.832,E2 -16981.832} C_VEL
LIN {X 0,Y 303.4,Z 386.131,A -85,B 0,C 180,E1 -16982.084,E2 -16982.084} C_VEL
LIN {X 0,Y 301.429,Z 444.331,A -85,B 0,C 180,E1 -16983.496,E2 -16983.496} C_VEL
LIN {X 0,Y 300.314,Z 457.205,A -85,B 0,C 180,E1 -16984.019,E2 -16984.019} C_VEL
LIN {X 0,Y 298.679,Z 470.577,A -85,B 0,C 180,E1 -16984.848,E2 -16984.848} C_VEL
LIN {X 0,Y 296.757,Z 482.633,A -85,B 0,C 180,E1 -16985.887,E2 -16985.887} C_VEL
LIN {X 0,Y 294.691,Z 494.098,A -85,B 0,C 180,E1 -16987.198,E2 -16987.198} C_VEL
LIN {X 0,Y 292.364,Z 504.465,A -85,B 0,C 180,E1 -16988.679,E2 -16988.679} C_VEL
LIN {X 0,Y 290.405,Z 512.953,A -85,B 0,C 180,E1 -16990.195,E2 -16990.195} C_VEL
LIN {X 0,Y 288.381,Z 521.484,A -85,B 0,C 180,E1 -16992.071,E2 -16992.071} C_VEL
LIN {X 0,Y 286.48,Z 529.636,A -85,B 0,C 180,E1 -16994.344,E2 -16994.344} C_VEL
LIN {X 0,Y 284.861,Z 535.643,A -85,B 0,C 180,E1 -16996.444,E2 -16996.444} C_VEL
LIN {X 0,Y 283.765,Z 540.419,A -85,B 0,C 180,E1 -16998.571,E2 -16998.571} C_VEL
LIN {X 0,Y 283.034,Z 544.102,A -85,B 0,C 180,E1 -17000.711,E2 -17000.711} C_VEL
LIN {X 0,Y 282.556,Z 546.792,A -85,B 0,C 180,E1 -17002.855,E2 -17002.855} C_VEL
LIN {X 0,Y 282.403,Z 548.277,A -85,B 0,C 180,E1 -17004.539,E2 -17004.539} C_VEL
LIN {X 0,Y 282.377,Z 549.428,A -85,B 0,C 180,E1 -17007.146,E2 -17007.146} C_VEL
LIN {X 0,Y 282.366,Z 549.495,A -85,B 0,C 180,E1 -17008.573,E2 -17008.573} C_VEL
LIN {X 0,Y 282.412,Z 549.177,A -85,B 0,C 180,E1 -17009.999,E2 -17009.999} C_VEL
LIN {X 0,Y 282.391,Z 548.466,A -85,B 0,C 180,E1 -17011.425,E2 -17011.425} C_VEL
LIN {X 0,Y 282.423,Z 547.312,A -85,B 0,C 180,E1 -17012.852,E2 -17012.852} C_VEL
LIN {X 0,Y 282.416,Z 544.053,A -85,B 0,C 180,E1 -17015.489,E2 -17015.489} C_VEL
LIN {X 0,Y 282.665,Z 539.808,A -85,B 0,C 180,E1 -17017.859,E2 -17017.859} C_VEL
LIN {X 0,Y 283.076,Z 534.738,A -85,B 0,C 180,E1 -17020.007,E2 -17020.007} C_VEL
LIN {X 0,Y 283.73,Z 528.344,A -85,B 0,C 180,E1 -17022.153,E2 -17022.153} C_VEL
LIN {X 0,Y 284.81,Z 520.323,A -85,B 0,C 180,E1 -17024.285,E2 -17024.285} C_VEL
LIN {X 0,Y 286.049,Z 511.161,A -85,B 0,C 180,E1 -17026.241,E2 -17026.241} C_VEL
LIN {X 0,Y 287.361,Z 501.002,A -85,B 0,C 180,E1 -17027.984,E2 -17027.984} C_VEL
LIN {X 0,Y 288.621,Z 490.839,A -85,B 0,C 180,E1 -17029.375,E2 -17029.375} C_VEL
LIN {X 0,Y 289.904,Z 479.769,A -85,B 0,C 180,E1 -17030.579,E2 -17030.579} C_VEL
LIN {X 0,Y 291.131,Z 467.51,A -85,B 0,C 180,E1 -17031.6,E2 -17031.6} C_VEL
LIN {X 0,Y 292.173,Z 454.725,A -85,B 0,C 180,E1 -17032.354,E2 -17032.354} C_VEL
LIN {X 0,Y 292.82,Z 440.97,A -85,B 0,C 180,E1 -17032.868,E2 -17032.868} C_VEL
LIN {X 0,Y 294.035,Z 380.541,A -85,B 0,C 180,E1 -17034.344,E2 -17034.344} C_VEL
LIN {X 0,Y 288.625,Z 339.878,A -85,B 0,C 180,E1 -17035.794,E2 -17035.794} C_VEL
LIN {X 0,Y 288.239,Z 336.716,A -85,B 0,C 180,E1 -17035.939,E2 -17035.939} C_VEL
LIN {X 0,Y 288.126,Z 333.679,A -85,B 0,C 180,E1 -17036.823,E2 -17036.823} C_VEL
LIN {X 0,Y 286.069,Z 323.017,A -85,B 0,C 180,E1 -17040.11,E2 -17040.11} C_VEL
LIN {X 0,Y 284.288,Z 315.074,A -85,B 0,C 180,E1 -17042.678,E2 -17042.678} C_VEL
LIN {X 0,Y 284.331,Z 315.068,A -85,B 0,C 180,E1 -17046.384,E2 -17046.384} C_VEL
LIN {X 0,Y 284.302,Z 315.069,A -85,B 0,C 180,E1 -17049.993,E2 -17049.993} C_VEL
LIN {X 0,Y 284.241,Z 315.079,A -85,B 0,C 180,E1 -17054.189,E2 -17054.189} C_VEL
LIN {X 0,Y 284.283,Z 315.073,A -85,B 0,C 180,E1 -17058.126,E2 -17058.126} C_VEL
LIN {X 0,Y 284.33,Z 315.066,A -85,B 0,C 180,E1 -17062.273,E2 -17062.273} C_VEL
LIN {X 0,Y 284.317,Z 315.067,A -85,B 0,C 180,E1 -17065.352,E2 -17065.352} C_VEL
LIN {X 0,Y 284.292,Z 315.072,A -85,B 0,C 180,E1 -17068.725,E2 -17068.725} C_VEL
LIN {X 0,Y 284.39,Z 315.06,A -85,B 0,C 180,E1 -17072.826,E2 -17072.826} C_VEL
LIN {X 0,Y 284.359,Z 315.062,A -85,B 0,C 180,E1 -17076.706,E2 -17076.706} C_VEL
LIN {X 0,Y 284.396,Z 315.054,A -85,B 0,C 180,E1 -17081.261,E2 -17081.261} C_VEL
LIN {X 0,Y 284.47,Z 315.042,A -85,B 0,C 180,E1 -17084.469,E2 -17084.469} C_VEL
LIN {X 0,Y 284.48,Z 315.046,A -85,B 0,C 180,E1 -17088.601,E2 -17088.601} C_VEL
LIN {X 0,Y 284.651,Z 315.023,A -85,B 0,C 180,E1 -17091.481,E2 -17091.481} C_VEL
LIN {X 0,Y 284.593,Z 315.022,A -85,B 0,C 180,E1 -17094.331,E2 -17094.331} C_VEL
LIN {X 0,Y 284.847,Z 314.999,A -85,B 0,C 180,E1 -17098.586,E2 -17098.586} C_VEL
LIN {X 0,Y 284.847,Z 315.002,A -85,B 0,C 180,E1 -17101.414,E2 -17101.414} C_VEL
LIN {X 0,Y 284.644,Z 315.016,A -85,B 0,C 180,E1 -17107.091,E2 -17107.091} C_VEL
LIN {X 0,Y 284.509,Z 315.044,A -85,B 0,C 180,E1 -17109.957,E2 -17109.957} C_VEL
LIN {X 0,Y 284.474,Z 315.047,A -85,B 0,C 180,E1 -17114.303,E2 -17114.303} C_VEL
LIN {X 0,Y 284.418,Z 315.053,A -85,B 0,C 180,E1 -17117.249,E2 -17117.249} C_VEL
LIN {X 0,Y 284.37,Z 315.063,A -85,B 0,C 180,E1 -17120.243,E2 -17120.243} C_VEL
LIN {X 0,Y 284.331,Z 315.066,A -85,B 0,C 180,E1 -17124.847,E2 -17124.847} C_VEL
LIN {X 0,Y 284.325,Z 315.065,A -85,B 0,C 180,E1 -17128.011,E2 -17128.011} C_VEL
LIN {X 0,Y 284.289,Z 315.069,A -85,B 0,C 180,E1 -17131.275,E2 -17131.275} C_VEL
LIN {X 0,Y 284.334,Z 315.064,A -85,B 0,C 180,E1 -17135.349,E2 -17135.349} C_VEL
LIN {X 0,Y 284.295,Z 315.069,A -85,B 0,C 180,E1 -17138.172,E2 -17138.172} C_VEL
LIN {X 0,Y 284.232,Z 315.077,A -85,B 0,C 180,E1 -17142.118,E2 -17142.118} C_VEL
LIN {X 0,Y 284.233,Z 315.077,A -85,B 0,C 180,E1 -17146.187,E2 -17146.187} C_VEL
LIN {X 0,Y 284.279,Z 315.071,A -85,B 0,C 180,E1 -17150.031,E2 -17150.031} C_VEL
LIN {X 0,Y 284.323,Z 315.067,A -85,B 0,C 180,E1 -17153.615,E2 -17153.615} C_VEL
LIN {X 0,Y 284.303,Z 315.072,A -85,B 0,C 180,E1 -17157.192,E2 -17157.192} C_VEL
LIN {X 0,Y 284.334,Z 315.063,A -85,B 0,C 180,E1 -17160.375,E2 -17160.375} C_VEL
LIN {X 0,Y 284.303,Z 315.072,A -85,B 0,C 180,E1 -17163.581,E2 -17163.581} C_VEL
LIN {X 0,Y 284.326,Z 315.066,A -85,B 0,C 180,E1 -17166.705,E2 -17166.705} C_VEL
LIN {X 0,Y 284.376,Z 315.062,A -85,B 0,C 180,E1 -17169.906,E2 -17169.906} C_VEL
LIN {X 0,Y 284.455,Z 315.051,A -85,B 0,C 180,E1 -17174.488,E2 -17174.488} C_VEL
LIN {X 0,Y 284.496,Z 315.188,A -85,B 0,C 180,E1 -17177.155,E2 -17177.155} C_VEL
LIN {X 0,Y 284.994,Z 317.535,A -85,B 0,C 180,E1 -17177.924,E2 -17177.924} C_VEL
LIN {X 0,Y 292.287,Z 337.896,A -85,B 0,C 180,E1 -17179.024,E2 -17179.024} C_VEL
LIN {X 0,Y 293.745,Z 343.322,A -85,B 0,C 180,E1 -17179.272,E2 -17179.272} C_VEL
LIN {X 0,Y 294.896,Z 350.427,A -85,B 0,C 180,E1 -17179.539,E2 -17179.539} C_VEL
LIN {X 0,Y 292.891,Z 424.727,A -85,B 0,C 180,E1 -17181.345,E2 -17181.345} C_VEL
LIN {X 0,Y 292.262,Z 437.681,A -85,B 0,C 180,E1 -17181.923,E2 -17181.923} C_VEL
LIN {X 0,Y 291.291,Z 450.989,A -85,B 0,C 180,E1 -17182.811,E2 -17182.811} C_VEL
LIN {X 0,Y 290.26,Z 462.929,A -85,B 0,C 180,E1 -17183.92,E2 -17183.92} C_VEL
LIN {X 0,Y 288.97,Z 474.381,A -85,B 0,C 180,E1 -17185.292,E2 -17185.292} C_VEL
LIN {X 0,Y 287.638,Z 484.722,A -85,B 0,C 180,E1 -17186.85,E2 -17186.85} C_VEL
LIN {X 0,Y 286.282,Z 494.015,A -85,B 0,C 180,E1 -17188.594,E2 -17188.594} C_VEL
LIN {X 0,Y 285.035,Z 503.013,A -85,B 0,C 180,E1 -17190.707,E2 -17190.707} C_VEL
LIN {X 0,Y 284.094,Z 510.26,A -85,B 0,C 180,E1 -17192.837,E2 -17192.837} C_VEL
LIN {X 0,Y 283.352,Z 516.051,A -85,B 0,C 180,E1 -17194.981,E2 -17194.981} C_VEL
LIN {X 0,Y 282.896,Z 520.603,A -85,B 0,C 180,E1 -17197.136,E2 -17197.136} C_VEL
LIN {X 0,Y 282.602,Z 523.015,A -85,B 0,C 180,E1 -17198.582,E2 -17198.582} C_VEL
LIN {X 0,Y 282.385,Z 524.994,A -85,B 0,C 180,E1 -17200.034,E2 -17200.034} C_VEL
LIN {X 0,Y 282.259,Z 526.541,A -85,B 0,C 180,E1 -17201.491,E2 -17201.491} C_VEL
LIN {X 0,Y 282.252,Z 528.092,A -85,B 0,C 180,E1 -17203.809,E2 -17203.809} C_VEL
LIN {X 0,Y 282.227,Z 528.598,A -85,B 0,C 180,E1 -17205.899,E2 -17205.899} C_VEL
LIN {X 0,Y 282.414,Z 528.445,A -85,B 0,C 180,E1 -17207.376,E2 -17207.376} C_VEL
LIN {X 0,Y 282.756,Z 527.685,A -85,B 0,C 180,E1 -17209.177,E2 -17209.177} C_VEL
LIN {X 0,Y 283.413,Z 525.435,A -85,B 0,C 180,E1 -17211.838,E2 -17211.838} C_VEL
LIN {X 0,Y 284.19,Z 522.82,A -85,B 0,C 180,E1 -17213.793,E2 -17213.793} C_VEL
LIN {X 0,Y 285.457,Z 518.195,A -85,B 0,C 180,E1 -17216.307,E2 -17216.307} C_VEL
LIN {X 0,Y 287.262,Z 511.743,A -85,B 0,C 180,E1 -17218.868,E2 -17218.868} C_VEL
LIN {X 0,Y 289.157,Z 504.576,A -85,B 0,C 180,E1 -17221.066,E2 -17221.066} C_VEL
LIN {X 0,Y 290.994,Z 497.006,A -85,B 0,C 180,E1 -17222.917,E2 -17222.917} C_VEL
LIN {X 0,Y 293.167,Z 487.874,A -85,B 0,C 180,E1 -17224.706,E2 -17224.706} C_VEL
LIN {X 0,Y 295.298,Z 478.024,A -85,B 0,C 180,E1 -17226.255,E2 -17226.255} C_VEL
LIN {X 0,Y 297.4,Z 466.493,A -85,B 0,C 180,E1 -17227.696,E2 -17227.696} C_VEL
LIN {X 0,Y 299.137,Z 454.694,A -85,B 0,C 180,E1 -17228.83,E2 -17228.83} C_VEL
LIN {X 0,Y 300.622,Z 441.6,A -85,B 0,C 180,E1 -17229.768,E2 -17229.768} C_VEL
LIN {X 0,Y 301.606,Z 428.602,A -85,B 0,C 180,E1 -17230.398,E2 -17230.398} C_VEL
LIN {X 0,Y 302.394,Z 412.029,A -85,B 0,C 180,E1 -17230.851,E2 -17230.851} C_VEL
LIN {X 0,Y 304.3,Z 356.433,A -85,B 0,C 180,E1 -17232.169,E2 -17232.169} C_VEL
LIN {X 0,Y 297.136,Z 340.525,A -85,B 0,C 180,E1 -17233.538,E2 -17233.538} C_VEL
LIN {X 0,Y 289.036,Z 325.444,A -85,B 0,C 180,E1 -17235.115,E2 -17235.115} C_VEL
LIN {X 0,Y 285.141,Z 318.258,A -85,B 0,C 180,E1 -17235.957,E2 -17235.957} C_VEL
LIN {X 0,Y 284.317,Z 315.064,A -85,B 0,C 180,E1 -17237.331,E2 -17237.331} C_VEL
LIN {X 0,Y 284.309,Z 315.059,A -85,B 0,C 180,E1 -17240.024,E2 -17240.024} C_VEL
LIN {X 0,Y 284.335,Z 315.068,A -85,B 0,C 180,E1 -17243.614,E2 -17243.614} C_VEL
LIN {X 0,Y 284.31,Z 315.066,A -85,B 0,C 180,E1 -17247.19,E2 -17247.19} C_VEL
LIN {X 0,Y 284.361,Z 315.057,A -85,B 0,C 180,E1 -17250.376,E2 -17250.376} C_VEL
LIN {X 0,Y 284.384,Z 315.054,A -85,B 0,C 180,E1 -17253.206,E2 -17253.206} C_VEL
LIN {X 0,Y 283.678,Z 315.146,A -85,B 0,C 180,E1 -17254.387,E2 -17254.387} C_VEL
LIN {X 0,Y 280.745,Z 315.517,A -85,B 0,C 180,E1 -17256.31,E2 -17256.31} C_VEL
LIN {X 0,Y 278.323,Z 315.821,A -85,B 0,C 180,E1 -17257.872,E2 -17257.872} C_VEL
LIN {X 0,Y 277.363,Z 315.936,A -85,B 0,C 180,E1 -17259.084,E2 -17259.084} C_VEL
LIN {X 0,Y 277.327,Z 315.938,A -85,B 0,C 180,E1 -17259.494,E2 -17259.494} C_VEL
LIN {X 0,Y 277.408,Z 315.927,A -85,B 0,C 180,E1 -17263.818,E2 -17263.818} C_VEL
LIN {X 0,Y 277.419,Z 315.922,A -85,B 0,C 180,E1 -17266.82,E2 -17266.82} C_VEL
LIN {X 0,Y 277.618,Z 315.891,A -85,B 0,C 180,E1 -17271.263,E2 -17271.263} C_VEL
LIN {X 0,Y 277.573,Z 315.904,A -85,B 0,C 180,E1 -17274.187,E2 -17274.187} C_VEL
LIN {X 0,Y 277.822,Z 315.876,A -85,B 0,C 180,E1 -17278.55,E2 -17278.55} C_VEL
LIN {X 0,Y 277.822,Z 315.861,A -85,B 0,C 180,E1 -17281.449,E2 -17281.449} C_VEL
LIN {X 0,Y 277.655,Z 315.889,A -85,B 0,C 180,E1 -17287.271,E2 -17287.271} C_VEL
LIN {X 0,Y 277.509,Z 315.905,A -85,B 0,C 180,E1 -17290.211,E2 -17290.211} C_VEL
LIN {X 0,Y 277.436,Z 315.92,A -85,B 0,C 180,E1 -17294.674,E2 -17294.674} C_VEL
LIN {X 0,Y 277.347,Z 315.935,A -85,B 0,C 180,E1 -17299.234,E2 -17299.234} C_VEL
LIN {X 0,Y 277.293,Z 315.944,A -85,B 0,C 180,E1 -17304.157,E2 -17304.157} C_VEL
LIN {X 0,Y 277.326,Z 315.94,A -85,B 0,C 180,E1 -17307.504,E2 -17307.504} C_VEL
LIN {X 0,Y 277.274,Z 315.935,A -85,B 0,C 180,E1 -17310.481,E2 -17310.481} C_VEL
LIN {X 0,Y 277.249,Z 315.939,A -85,B 0,C 180,E1 -17313.896,E2 -17313.896} C_VEL
LIN {X 0,Y 277.269,Z 315.94,A -85,B 0,C 180,E1 -17317.469,E2 -17317.469} C_VEL
LIN {X 0,Y 277.212,Z 315.951,A -85,B 0,C 180,E1 -17321.236,E2 -17321.236} C_VEL
LIN {X 0,Y 277.203,Z 315.955,A -85,B 0,C 180,E1 -17325.226,E2 -17325.226} C_VEL
LIN {X 0,Y 277.225,Z 315.95,A -85,B 0,C 180,E1 -17329.512,E2 -17329.512} C_VEL
LIN {X 0,Y 277.301,Z 316.096,A -85,B 0,C 180,E1 -17330.137,E2 -17330.137} C_VEL
LIN {X 0,Y 279.871,Z 325.257,A -85,B 0,C 180,E1 -17333.927,E2 -17333.927} C_VEL
LIN {X 0,Y 282.288,Z 335.261,A -85,B 0,C 180,E1 -17337.714,E2 -17337.714} C_VEL
LIN {X 0,Y 284.415,Z 339.542,A -85,B 0,C 180,E1 -17338.173,E2 -17338.173} C_VEL
LIN {X 0,Y 291.91,Z 355.53,A -85,B 0,C 180,E1 -17339.734,E2 -17339.734} C_VEL
LIN {X 0,Y 295.307,Z 372.173,A -85,B 0,C 180,E1 -17340.678,E2 -17340.678} C_VEL
LIN {X 0,Y 297.423,Z 386.46,A -85,B 0,C 180,E1 -17341.361,E2 -17341.361} C_VEL
LIN {X 0,Y 295.338,Z 444.498,A -85,B 0,C 180,E1 -17342.795,E2 -17342.795} C_VEL
LIN {X 0,Y 294.089,Z 458.188,A -85,B 0,C 180,E1 -17343.379,E2 -17343.379} C_VEL
LIN {X 0,Y 292.485,Z 470.677,A -85,B 0,C 180,E1 -17344.181,E2 -17344.181} C_VEL
LIN {X 0,Y 290.649,Z 481.836,A -85,B 0,C 180,E1 -17345.156,E2 -17345.156} C_VEL
LIN {X 0,Y 288.455,Z 493.402,A -85,B 0,C 180,E1 -17346.486,E2 -17346.486} C_VEL
LIN {X 0,Y 286.046,Z 503.841,A -85,B 0,C 180,E1 -17347.994,E2 -17347.994} C_VEL
LIN {X 0,Y 283.747,Z 513.271,A -85,B 0,C 180,E1 -17349.71,E2 -17349.71} C_VEL
LIN {X 0,Y 281.514,Z 522.13,A -85,B 0,C 180,E1 -17351.748,E2 -17351.748} C_VEL
LIN {X 0,Y 279.627,Z 529.733,A -85,B 0,C 180,E1 -17353.95,E2 -17353.95} C_VEL
LIN {X 0,Y 277.948,Z 535.668,A -85,B 0,C 180,E1 -17356.1,E2 -17356.1} C_VEL
LIN {X 0,Y 276.784,Z 540.378,A -85,B 0,C 180,E1 -17358.279,E2 -17358.279} C_VEL
LIN {X 0,Y 275.994,Z 544.003,A -85,B 0,C 180,E1 -17360.472,E2 -17360.472} C_VEL
LIN {X 0,Y 275.494,Z 546.64,A -85,B 0,C 180,E1 -17362.671,E2 -17362.671} C_VEL
LIN {X 0,Y 275.321,Z 548.19,A -85,B 0,C 180,E1 -17364.585,E2 -17364.585} C_VEL
LIN {X 0,Y 275.284,Z 549.174,A -85,B 0,C 180,E1 -17367.072,E2 -17367.072} C_VEL
LIN {X 0,Y 275.29,Z 549.217,A -85,B 0,C 180,E1 -17368.536,E2 -17368.536} C_VEL
LIN {X 0,Y 275.331,Z 548.874,A -85,B 0,C 180,E1 -17369.999,E2 -17369.999} C_VEL
LIN {X 0,Y 275.314,Z 548.126,A -85,B 0,C 180,E1 -17371.462,E2 -17371.462} C_VEL
LIN {X 0,Y 275.329,Z 546.931,A -85,B 0,C 180,E1 -17372.925,E2 -17372.925} C_VEL
LIN {X 0,Y 275.331,Z 543.904,A -85,B 0,C 180,E1 -17375.436,E2 -17375.436} C_VEL
LIN {X 0,Y 275.589,Z 539.314,A -85,B 0,C 180,E1 -17378.062,E2 -17378.062} C_VEL
LIN {X 0,Y 276.135,Z 533.178,A -85,B 0,C 180,E1 -17380.632,E2 -17380.632} C_VEL
LIN {X 0,Y 276.913,Z 526.442,A -85,B 0,C 180,E1 -17382.83,E2 -17382.83} C_VEL
LIN {X 0,Y 278.063,Z 518.072,A -85,B 0,C 180,E1 -17385.013,E2 -17385.013} C_VEL
LIN {X 0,Y 279.232,Z 509.509,A -85,B 0,C 180,E1 -17386.813,E2 -17386.813} C_VEL
LIN {X 0,Y 280.67,Z 498.788,A -85,B 0,C 180,E1 -17388.617,E2 -17388.617} C_VEL
LIN {X 0,Y 281.852,Z 489.654,A -85,B 0,C 180,E1 -17389.86,E2 -17389.86} C_VEL
LIN {X 0,Y 283.203,Z 478.367,A -85,B 0,C 180,E1 -17391.089,E2 -17391.089} C_VEL
LIN {X 0,Y 284.397,Z 466.94,A -85,B 0,C 180,E1 -17392.042,E2 -17392.042} C_VEL
LIN {X 0,Y 285.47,Z 453.966,A -85,B 0,C 180,E1 -17392.813,E2 -17392.813} C_VEL
LIN {X 0,Y 286.095,Z 440.252,A -85,B 0,C 180,E1 -17393.329,E2 -17393.329} C_VEL
LIN {X 0,Y 287.388,Z 381.669,A -85,B 0,C 180,E1 -17394.786,E2 -17394.786} C_VEL
LIN {X 0,Y 282.117,Z 341.491,A -85,B 0,C 180,E1 -17396.257,E2 -17396.257} C_VEL
LIN {X 0,Y 281.344,Z 336.495,A -85,B 0,C 180,E1 -17396.475,E2 -17396.475} C_VEL
LIN {X 0,Y 280.005,Z 328.742,A -85,B 0,C 180,E1 -17398.89,E2 -17398.89} C_VEL
LIN {X 0,Y 277.626,Z 317.727,A -85,B 0,C 180,E1 -17402.473,E2 -17402.473} C_VEL
LIN {X 0,Y 277.249,Z 315.95,A -85,B 0,C 180,E1 -17403.097,E2 -17403.097} C_VEL
LIN {X 0,Y 277.278,Z 315.945,A -85,B 0,C 180,E1 -17405.798,E2 -17405.798} C_VEL
LIN {X 0,Y 277.233,Z 315.948,A -85,B 0,C 180,E1 -17409.326,E2 -17409.326} C_VEL
LIN {X 0,Y 277.205,Z 315.953,A -85,B 0,C 180,E1 -17413.197,E2 -17413.197} C_VEL
LIN {X 0,Y 277.217,Z 315.952,A -85,B 0,C 180,E1 -17417.322,E2 -17417.322} C_VEL
LIN {X 0,Y 277.27,Z 315.943,A -85,B 0,C 180,E1 -17421.789,E2 -17421.789} C_VEL
LIN {X 0,Y 277.297,Z 315.942,A -85,B 0,C 180,E1 -17424.343,E2 -17424.343} C_VEL
LIN {X 0,Y 277.24,Z 315.946,A -85,B 0,C 180,E1 -17427.836,E2 -17427.836} C_VEL
LIN {X 0,Y 277.283,Z 315.944,A -85,B 0,C 180,E1 -17431.212,E2 -17431.212} C_VEL
LIN {X 0,Y 277.307,Z 315.941,A -85,B 0,C 180,E1 -17434.479,E2 -17434.479} C_VEL
LIN {X 0,Y 277.278,Z 315.944,A -85,B 0,C 180,E1 -17437.654,E2 -17437.654} C_VEL
LIN {X 0,Y 277.337,Z 315.936,A -85,B 0,C 180,E1 -17440.766,E2 -17440.766} C_VEL
LIN {X 0,Y 277.42,Z 315.926,A -85,B 0,C 180,E1 -17445.325,E2 -17445.325} C_VEL
LIN {X 0,Y 277.499,Z 315.916,A -85,B 0,C 180,E1 -17449.788,E2 -17449.788} C_VEL
LIN {X 0,Y 277.645,Z 315.891,A -85,B 0,C 180,E1 -17452.729,E2 -17452.729} C_VEL
LIN {X 0,Y 277.813,Z 315.875,A -85,B 0,C 180,E1 -17458.55,E2 -17458.55} C_VEL
LIN {X 0,Y 277.813,Z 315.879,A -85,B 0,C 180,E1 -17461.45,E2 -17461.45} C_VEL
LIN {X 0,Y 277.602,Z 315.892,A -85,B 0,C 180,E1 -17467.272,E2 -17467.272} C_VEL
LIN {X 0,Y 277.452,Z 315.924,A -85,B 0,C 180,E1 -17470.213,E2 -17470.213} C_VEL
LIN {X 0,Y 277.427,Z 315.923,A -85,B 0,C 180,E1 -17474.675,E2 -17474.675} C_VEL
LIN {X 0,Y 277.337,Z 315.936,A -85,B 0,C 180,E1 -17479.235,E2 -17479.235} C_VEL
LIN {X 0,Y 277.285,Z 315.945,A -85,B 0,C 180,E1 -17484.159,E2 -17484.159} C_VEL
LIN {X 0,Y 277.319,Z 315.935,A -85,B 0,C 180,E1 -17487.506,E2 -17487.506} C_VEL
LIN {X 0,Y 277.266,Z 315.949,A -85,B 0,C 180,E1 -17490.482,E2 -17490.482} C_VEL
LIN {X 0,Y 277.241,Z 315.945,A -85,B 0,C 180,E1 -17493.897,E2 -17493.897} C_VEL
LIN {X 0,Y 277.254,Z 315.945,A -85,B 0,C 180,E1 -17497.472,E2 -17497.472} C_VEL
LIN {X 0,Y 277.178,Z 315.957,A -85,B 0,C 180,E1 -17501.242,E2 -17501.242} C_VEL
LIN {X 0,Y 277.169,Z 315.959,A -85,B 0,C 180,E1 -17505.234,E2 -17505.234} C_VEL
LIN {X 0,Y 277.18,Z 315.958,A -85,B 0,C 180,E1 -17508.76,E2 -17508.76} C_VEL
LIN {X 0,Y 277.257,Z 315.947,A -85,B 0,C 180,E1 -17512.531,E2 -17512.531} C_VEL
LIN {X 0,Y 277.243,Z 315.947,A -85,B 0,C 180,E1 -17516.106,E2 -17516.106} C_VEL
LIN {X 0,Y 277.26,Z 315.947,A -85,B 0,C 180,E1 -17519.54,E2 -17519.54} C_VEL
LIN {X 0,Y 277.289,Z 315.944,A -85,B 0,C 180,E1 -17522.858,E2 -17522.858} C_VEL
LIN {X 0,Y 277.281,Z 315.944,A -85,B 0,C 180,E1 -17526.077,E2 -17526.077} C_VEL
LIN {X 0,Y 277.324,Z 315.939,A -85,B 0,C 180,E1 -17530.766,E2 -17530.766} C_VEL
LIN {X 0,Y 277.414,Z 315.93,A -85,B 0,C 180,E1 -17535.326,E2 -17535.326} C_VEL
LIN {X 0,Y 277.429,Z 315.973,A -85,B 0,C 180,E1 -17536.729,E2 -17536.729} C_VEL
LIN {X 0,Y 277.773,Z 317.692,A -85,B 0,C 180,E1 -17537.329,E2 -17537.329} C_VEL
LIN {X 0,Y 284.893,Z 337.199,A -85,B 0,C 180,E1 -17538.445,E2 -17538.445} C_VEL
LIN {X 0,Y 287.162,Z 344.678,A -85,B 0,C 180,E1 -17538.819,E2 -17538.819} C_VEL
LIN {X 0,Y 288.251,Z 350.805,A -85,B 0,C 180,E1 -17539.063,E2 -17539.063} C_VEL
LIN {X 0,Y 286.171,Z 425.04,A -85,B 0,C 180,E1 -17540.905,E2 -17540.905} C_VEL
LIN {X 0,Y 285.499,Z 438.195,A -85,B 0,C 180,E1 -17541.508,E2 -17541.508} C_VEL
LIN {X 0,Y 284.538,Z 450.882,A -85,B 0,C 180,E1 -17542.372,E2 -17542.372} C_VEL
LIN {X 0,Y 283.564,Z 461.835,A -85,B 0,C 180,E1 -17543.385,E2 -17543.385} C_VEL
LIN {X 0,Y 282.244,Z 473.657,A -85,B 0,C 180,E1 -17544.804,E2 -17544.804} C_VEL
LIN {X 0,Y 280.808,Z 484.282,A -85,B 0,C 180,E1 -17546.414,E2 -17546.414} C_VEL
LIN {X 0,Y 279.428,Z 493.733,A -85,B 0,C 180,E1 -17548.199,E2 -17548.199} C_VEL
LIN {X 0,Y 278.104,Z 502.826,A -85,B 0,C 180,E1 -17550.363,E2 -17550.363} C_VEL
LIN {X 0,Y 277.09,Z 510.155,A -85,B 0,C 180,E1 -17552.545,E2 -17552.545} C_VEL
LIN {X 0,Y 276.399,Z 515.122,A -85,B 0,C 180,E1 -17554.376,E2 -17554.376} C_VEL
LIN {X 0,Y 275.92,Z 519.961,A -85,B 0,C 180,E1 -17556.596,E2 -17556.596} C_VEL
LIN {X 0,Y 275.456,Z 523.646,A -85,B 0,C 180,E1 -17558.807,E2 -17558.807} C_VEL
LIN {X 0,Y 275.252,Z 525.565,A -85,B 0,C 180,E1 -17560.297,E2 -17560.297} C_VEL
LIN {X 0,Y 275.161,Z 527.003,A -85,B 0,C 180,E1 -17561.791,E2 -17561.791} C_VEL
LIN {X 0,Y 275.161,Z 528.364,A -85,B 0,C 180,E1 -17563.932,E2 -17563.932} C_VEL
LIN {X 0,Y 275.187,Z 528.871,A -85,B 0,C 180,E1 -17566.317,E2 -17566.317} C_VEL
LIN {X 0,Y 275.394,Z 528.633,A -85,B 0,C 180,E1 -17567.833,E2 -17567.833} C_VEL
LIN {X 0,Y 275.713,Z 527.959,A -85,B 0,C 180,E1 -17569.414,E2 -17569.414} C_VEL
LIN {X 0,Y 276.037,Z 526.938,A -85,B 0,C 180,E1 -17570.883,E2 -17570.883} C_VEL
LIN {X 0,Y 276.517,Z 525.398,A -85,B 0,C 180,E1 -17572.411,E2 -17572.411} C_VEL
LIN {X 0,Y 277.538,Z 522.214,A -85,B 0,C 180,E1 -17574.71,E2 -17574.71} C_VEL
LIN {X 0,Y 278.771,Z 517.909,A -85,B 0,C 180,E1 -17576.988,E2 -17576.988} C_VEL
LIN {X 0,Y 280.449,Z 512.296,A -85,B 0,C 180,E1 -17579.254,E2 -17579.254} C_VEL
LIN {X 0,Y 282.422,Z 505.191,A -85,B 0,C 180,E1 -17581.506,E2 -17581.506} C_VEL
LIN {X 0,Y 284.325,Z 497.842,A -85,B 0,C 180,E1 -17583.366,E2 -17583.366} C_VEL
LIN {X 0,Y 286.821,Z 487.82,A -85,B 0,C 180,E1 -17585.373,E2 -17585.373} C_VEL
LIN {X 0,Y 289.218,Z 477.263,A -85,B 0,C 180,E1 -17587.041,E2 -17587.041} C_VEL
LIN {X 0,Y 291.261,Z 466.244,A -85,B 0,C 180,E1 -17588.414,E2 -17588.414} C_VEL
LIN {X 0,Y 293.104,Z 454.094,A -85,B 0,C 180,E1 -17589.586,E2 -17589.586} C_VEL
LIN {X 0,Y 294.518,Z 442.113,A -85,B 0,C 180,E1 -17590.449,E2 -17590.449} C_VEL
LIN {X 0,Y 295.514,Z 429.775,A -85,B 0,C 180,E1 -17591.071,E2 -17591.071} C_VEL
LIN {X 0,Y 296.224,Z 414.703,A -85,B 0,C 180,E1 -17591.516,E2 -17591.516} C_VEL
LIN {X 0,Y 298.285,Z 358.396,A -85,B 0,C 180,E1 -17592.87,E2 -17592.87} C_VEL
LIN {X 0,Y 291.505,Z 343.421,A -85,B 0,C 180,E1 -17594.22,E2 -17594.22} C_VEL
LIN {X 0,Y 284.026,Z 329.434,A -85,B 0,C 180,E1 -17595.739,E2 -17595.739} C_VEL
LIN {X 0,Y 279.526,Z 321.632,A -85,B 0,C 180,E1 -17596.692,E2 -17596.692} C_VEL
LIN {X 0,Y 278.005,Z 318.622,A -85,B 0,C 180,E1 -17597.067,E2 -17597.067} C_VEL
LIN {X 0,Y 277.223,Z 315.958,A -85,B 0,C 180,E1 -17598.228,E2 -17598.228} C_VEL
LIN {X 0,Y 277.27,Z 315.948,A -85,B 0,C 180,E1 -17602.531,E2 -17602.531} C_VEL
LIN {X 0,Y 277.25,Z 315.95,A -85,B 0,C 180,E1 -17606.104,E2 -17606.104} C_VEL
LIN {X 0,Y 277.264,Z 315.941,A -85,B 0,C 180,E1 -17609.539,E2 -17609.539} C_VEL
LIN {X 0,Y 277.335,Z 315.931,A -85,B 0,C 180,E1 -17613.185,E2 -17613.185} C_VEL
LIN {X 0,Y 277.331,Z 315.935,A -85,B 0,C 180,E1 -17616.08,E2 -17616.08} C_VEL
LIN {X 0,Y 277.327,Z 315.938,A -85,B 0,C 180,E1 -17619.494,E2 -17619.494} C_VEL
LIN {X 0,Y 277.096,Z 315.962,A -85,B 0,C 180,E1 -17620.305,E2 -17620.305} C_VEL
LIN {X 0,Y 275.819,Z 316.123,A -85,B 0,C 180,E1 -17621.504,E2 -17621.504} C_VEL
LIN {X 0,Y 271.502,Z 316.661,A -85,B 0,C 180,E1 -17624.291,E2 -17624.291} C_VEL
LIN {X 0,Y 270.441,Z 316.785,A -85,B 0,C 180,E1 -17625.536,E2 -17625.536} C_VEL
LIN {X 0,Y 270.354,Z 316.796,A -85,B 0,C 180,E1 -17625.959,E2 -17625.959} C_VEL
LIN {X 0,Y 270.58,Z 316.765,A -85,B 0,C 180,E1 -17630.754,E2 -17630.754} C_VEL
LIN {X 0,Y 270.544,Z 316.78,A -85,B 0,C 180,E1 -17634.036,E2 -17634.036} C_VEL
LIN {X 0,Y 270.788,Z 316.752,A -85,B 0,C 180,E1 -17638.513,E2 -17638.513} C_VEL
LIN {X 0,Y 270.788,Z 316.737,A -85,B 0,C 180,E1 -17641.487,E2 -17641.487} C_VEL
LIN {X 0,Y 270.613,Z 316.767,A -85,B 0,C 180,E1 -17647.461,E2 -17647.461} C_VEL
LIN {X 0,Y 270.444,Z 316.782,A -85,B 0,C 180,E1 -17650.481,E2 -17650.481} C_VEL
LIN {X 0,Y 270.405,Z 316.794,A -85,B 0,C 180,E1 -17655.064,E2 -17655.064} C_VEL
LIN {X 0,Y 270.303,Z 316.811,A -85,B 0,C 180,E1 -17659.755,E2 -17659.755} C_VEL
LIN {X 0,Y 270.24,Z 316.816,A -85,B 0,C 180,E1 -17664.589,E2 -17664.589} C_VEL
LIN {X 0,Y 270.274,Z 316.818,A -85,B 0,C 180,E1 -17667.908,E2 -17667.908} C_VEL
LIN {X 0,Y 270.187,Z 316.826,A -85,B 0,C 180,E1 -17671.348,E2 -17671.348} C_VEL
LIN {X 0,Y 270.204,Z 316.821,A -85,B 0,C 180,E1 -17674.905,E2 -17674.905} C_VEL
LIN {X 0,Y 270.2,Z 316.827,A -85,B 0,C 180,E1 -17678.71,E2 -17678.71} C_VEL
LIN {X 0,Y 270.167,Z 316.828,A -85,B 0,C 180,E1 -17683.249,E2 -17683.249} C_VEL
LIN {X 0,Y 270.174,Z 316.83,A -85,B 0,C 180,E1 -17687.441,E2 -17687.441} C_VEL
LIN {X 0,Y 270.208,Z 316.973,A -85,B 0,C 180,E1 -17689.1,E2 -17689.1} C_VEL
LIN {X 0,Y 272.781,Z 325.975,A -85,B 0,C 180,E1 -17693.006,E2 -17693.006} C_VEL
LIN {X 0,Y 274.998,Z 334.839,A -85,B 0,C 180,E1 -17696.522,E2 -17696.522} C_VEL
LIN {X 0,Y 277.192,Z 339.252,A -85,B 0,C 180,E1 -17697.042,E2 -17697.042} C_VEL
LIN {X 0,Y 283.749,Z 352.603,A -85,B 0,C 180,E1 -17698.482,E2 -17698.482} C_VEL
LIN {X 0,Y 286.743,Z 359.65,A -85,B 0,C 180,E1 -17699.135,E2 -17699.135} C_VEL
LIN {X 0,Y 290.761,Z 381.585,A -85,B 0,C 180,E1 -17700.351,E2 -17700.351} C_VEL
LIN {X 0,Y 291.496,Z 387.426,A -85,B 0,C 180,E1 -17700.623,E2 -17700.623} C_VEL
LIN {X 0,Y 289.297,Z 444.323,A -85,B 0,C 180,E1 -17702.05,E2 -17702.05} C_VEL
LIN {X 0,Y 288.075,Z 457.679,A -85,B 0,C 180,E1 -17702.63,E2 -17702.63} C_VEL
LIN {X 0,Y 286.324,Z 470.773,A -85,B 0,C 180,E1 -17703.485,E2 -17703.485} C_VEL
LIN {X 0,Y 284.248,Z 482.616,A -85,B 0,C 180,E1 -17704.557,E2 -17704.557} C_VEL
LIN {X 0,Y 282.001,Z 493.988,A -85,B 0,C 180,E1 -17705.914,E2 -17705.914} C_VEL
LIN {X 0,Y 279.513,Z 504.282,A -85,B 0,C 180,E1 -17707.452,E2 -17707.452} C_VEL
LIN {X 0,Y 277.109,Z 513.555,A -85,B 0,C 180,E1 -17709.202,E2 -17709.202} C_VEL
LIN {X 0,Y 274.652,Z 522.785,A -85,B 0,C 180,E1 -17711.41,E2 -17711.41} C_VEL
LIN {X 0,Y 272.792,Z 529.838,A -85,B 0,C 180,E1 -17713.536,E2 -17713.536} C_VEL
LIN {X 0,Y 271.05,Z 535.702,A -85,B 0,C 180,E1 -17715.739,E2 -17715.739} C_VEL
LIN {X 0,Y 269.795,Z 540.348,A -85,B 0,C 180,E1 -17717.971,E2 -17717.971} C_VEL
LIN {X 0,Y 268.974,Z 543.912,A -85,B 0,C 180,E1 -17720.221,E2 -17720.221} C_VEL
LIN {X 0,Y 268.42,Z 546.492,A -85,B 0,C 180,E1 -17722.477,E2 -17722.477} C_VEL
LIN {X 0,Y 268.217,Z 548.124,A -85,B 0,C 180,E1 -17724.686,E2 -17724.686} C_VEL
LIN {X 0,Y 268.193,Z 548.922,A -85,B 0,C 180,E1 -17726.995,E2 -17726.995} C_VEL
LIN {X 0,Y 268.215,Z 548.94,A -85,B 0,C 180,E1 -17728.497,E2 -17728.497} C_VEL
LIN {X 0,Y 268.253,Z 548.572,A -85,B 0,C 180,E1 -17729.999,E2 -17729.999} C_VEL
LIN {X 0,Y 268.238,Z 547.775,A -85,B 0,C 180,E1 -17731.5,E2 -17731.5} C_VEL
LIN {X 0,Y 268.236,Z 546.551,A -85,B 0,C 180,E1 -17733.003,E2 -17733.003} C_VEL
LIN {X 0,Y 268.229,Z 543.811,A -85,B 0,C 180,E1 -17735.341,E2 -17735.341} C_VEL
LIN {X 0,Y 268.44,Z 540.265,A -85,B 0,C 180,E1 -17737.521,E2 -17737.521} C_VEL
LIN {X 0,Y 268.81,Z 535.46,A -85,B 0,C 180,E1 -17739.783,E2 -17739.783} C_VEL
LIN {X 0,Y 269.431,Z 529.365,A -85,B 0,C 180,E1 -17742.044,E2 -17742.044} C_VEL
LIN {X 0,Y 270.574,Z 521.783,A -85,B 0,C 180,E1 -17744.284,E2 -17744.284} C_VEL
LIN {X 0,Y 271.745,Z 514.025,A -85,B 0,C 180,E1 -17746.141,E2 -17746.141} C_VEL
LIN {X 0,Y 272.974,Z 504.528,A -85,B 0,C 180,E1 -17747.995,E2 -17747.995} C_VEL
LIN {X 0,Y 274.301,Z 493.951,A -85,B 0,C 180,E1 -17749.649,E2 -17749.649} C_VEL
LIN {X 0,Y 275.971,Z 482.241,A -85,B 0,C 180,E1 -17751.081,E2 -17751.081} C_VEL
LIN {X 0,Y 277.365,Z 469.735,A -85,B 0,C 180,E1 -17752.239,E2 -17752.239} C_VEL
LIN {X 0,Y 278.456,Z 457.307,A -85,B 0,C 180,E1 -17753.077,E2 -17753.077} C_VEL
LIN {X 0,Y 279.231,Z 444.743,A -85,B 0,C 180,E1 -17753.648,E2 -17753.648} C_VEL
LIN {X 0,Y 280.728,Z 382.573,A -85,B 0,C 180,E1 -17755.251,E2 -17755.251} C_VEL
LIN {X 0,Y 275.636,Z 343.173,A -85,B 0,C 180,E1 -17756.735,E2 -17756.735} C_VEL
LIN {X 0,Y 274.534,Z 337.582,A -85,B 0,C 180,E1 -17756.981,E2 -17756.981} C_VEL
LIN {X 0,Y 274.207,Z 336.276,A -85,B 0,C 180,E1 -17757.051,E2 -17757.051} C_VEL
LIN {X 0,Y 272.018,Z 325.101,A -85,B 0,C 180,E1 -17760.68,E2 -17760.68} C_VEL
LIN {X 0,Y 270.2,Z 316.828,A -85,B 0,C 180,E1 -17763.531,E2 -17763.531} C_VEL
LIN {X 0,Y 270.216,Z 316.824,A -85,B 0,C 180,E1 -17766.739,E2 -17766.739} C_VEL
LIN {X 0,Y 270.165,Z 316.829,A -85,B 0,C 180,E1 -17771.027,E2 -17771.027} C_VEL
LIN {X 0,Y 270.147,Z 316.832,A -85,B 0,C 180,E1 -17775.379,E2 -17775.379} C_VEL
LIN {X 0,Y 270.177,Z 316.826,A -85,B 0,C 180,E1 -17779.435,E2 -17779.435} C_VEL
LIN {X 0,Y 270.249,Z 316.818,A -85,B 0,C 180,E1 -17783.721,E2 -17783.721} C_VEL
LIN {X 0,Y 270.199,Z 316.827,A -85,B 0,C 180,E1 -17786.892,E2 -17786.892} C_VEL
LIN {X 0,Y 270.222,Z 316.823,A -85,B 0,C 180,E1 -17790.386,E2 -17790.386} C_VEL
LIN {X 0,Y 270.257,Z 316.818,A -85,B 0,C 180,E1 -17793.763,E2 -17793.763} C_VEL
LIN {X 0,Y 270.226,Z 316.826,A -85,B 0,C 180,E1 -17797.038,E2 -17797.038} C_VEL
LIN {X 0,Y 270.294,Z 316.811,A -85,B 0,C 180,E1 -17800.244,E2 -17800.244} C_VEL
LIN {X 0,Y 270.389,Z 316.797,A -85,B 0,C 180,E1 -17804.935,E2 -17804.935} C_VEL
LIN {X 0,Y 270.434,Z 316.798,A -85,B 0,C 180,E1 -17809.519,E2 -17809.519} C_VEL
LIN {X 0,Y 270.603,Z 316.767,A -85,B 0,C 180,E1 -17812.539,E2 -17812.539} C_VEL
LIN {X 0,Y 270.779,Z 316.752,A -85,B 0,C 180,E1 -17818.513,E2 -17818.513} C_VEL
LIN {X 0,Y 270.779,Z 316.755,A -85,B 0,C 180,E1 -17821.487,E2 -17821.487} C_VEL
LIN {X 0,Y 270.562,Z 316.769,A -85,B 0,C 180,E1 -17827.463,E2 -17827.463} C_VEL
LIN {X 0,Y 270.404,Z 316.8,A -85,B 0,C 180,E1 -17830.483,E2 -17830.483} C_VEL
LIN {X 0,Y 270.395,Z 316.798,A -85,B 0,C 180,E1 -17835.065,E2 -17835.065} C_VEL
LIN {X 0,Y 270.294,Z 316.815,A -85,B 0,C 180,E1 -17839.756,E2 -17839.756} C_VEL
LIN {X 0,Y 270.231,Z 316.824,A -85,B 0,C 180,E1 -17844.59,E2 -17844.59} C_VEL
LIN {X 0,Y 270.266,Z 316.815,A -85,B 0,C 180,E1 -17847.909,E2 -17847.909} C_VEL
LIN {X 0,Y 270.178,Z 316.827,A -85,B 0,C 180,E1 -17851.349,E2 -17851.349} C_VEL
LIN {X 0,Y 270.195,Z 316.827,A -85,B 0,C 180,E1 -17854.907,E2 -17854.907} C_VEL
LIN {X 0,Y 270.192,Z 316.827,A -85,B 0,C 180,E1 -17858.712,E2 -17858.712} C_VEL
LIN {X 0,Y 270.143,Z 316.831,A -85,B 0,C 180,E1 -17863.246,E2 -17863.246} C_VEL
LIN {X 0,Y 270.147,Z 316.832,A -85,B 0,C 180,E1 -17867.439,E2 -17867.439} C_VEL
LIN {X 0,Y 270.204,Z 316.827,A -85,B 0,C 180,E1 -17871.376,E2 -17871.376} C_VEL
LIN {X 0,Y 270.196,Z 316.83,A -85,B 0,C 180,E1 -17875.096,E2 -17875.096} C_VEL
LIN {X 0,Y 270.182,Z 316.832,A -85,B 0,C 180,E1 -17879.138,E2 -17879.138} C_VEL
LIN {X 0,Y 270.22,Z 316.823,A -85,B 0,C 180,E1 -17882.164,E2 -17882.164} C_VEL
LIN {X 0,Y 270.226,Z 316.825,A -85,B 0,C 180,E1 -17885.544,E2 -17885.544} C_VEL
LIN {X 0,Y 270.26,Z 316.819,A -85,B 0,C 180,E1 -17890.243,E2 -17890.243} C_VEL
LIN {X 0,Y 270.373,Z 316.806,A -85,B 0,C 180,E1 -17894.935,E2 -17894.935} C_VEL
LIN {X 0,Y 270.409,Z 316.887,A -85,B 0,C 180,E1 -17896.33,E2 -17896.33} C_VEL
LIN {X 0,Y 270.625,Z 317.981,A -85,B 0,C 180,E1 -17896.721,E2 -17896.721} C_VEL
LIN {X 0,Y 278.422,Z 339.119,A -85,B 0,C 180,E1 -17897.981,E2 -17897.981} C_VEL
LIN {X 0,Y 280.669,Z 346.319,A -85,B 0,C 180,E1 -17898.359,E2 -17898.359} C_VEL
LIN {X 0,Y 281.57,Z 351.178,A -85,B 0,C 180,E1 -17898.562,E2 -17898.562} C_VEL
LIN {X 0,Y 279.424,Z 425.576,A -85,B 0,C 180,E1 -17900.455,E2 -17900.455} C_VEL
LIN {X 0,Y 278.7,Z 439.385,A -85,B 0,C 180,E1 -17901.116,E2 -17901.116} C_VEL
LIN {X 0,Y 277.705,Z 451.822,A -85,B 0,C 180,E1 -17902,E2 -17902} C_VEL
LIN {X 0,Y 276.597,Z 463.689,A -85,B 0,C 180,E1 -17903.162,E2 -17903.162} C_VEL
LIN {X 0,Y 275.221,Z 475.235,A -85,B 0,C 180,E1 -17904.618,E2 -17904.618} C_VEL
LIN {X 0,Y 273.724,Z 485.908,A -85,B 0,C 180,E1 -17906.321,E2 -17906.321} C_VEL
LIN {X 0,Y 272.296,Z 495.072,A -85,B 0,C 180,E1 -17908.152,E2 -17908.152} C_VEL
LIN {X 0,Y 270.97,Z 503.985,A -85,B 0,C 180,E1 -17910.373,E2 -17910.373} C_VEL
LIN {X 0,Y 269.958,Z 511.144,A -85,B 0,C 180,E1 -17912.612,E2 -17912.612} C_VEL
LIN {X 0,Y 269.127,Z 517.659,A -85,B 0,C 180,E1 -17915.245,E2 -17915.245} C_VEL
LIN {X 0,Y 268.63,Z 521.972,A -85,B 0,C 180,E1 -17917.518,E2 -17917.518} C_VEL
LIN {X 0,Y 268.33,Z 524.27,A -85,B 0,C 180,E1 -17919.042,E2 -17919.042} C_VEL
LIN {X 0,Y 268.123,Z 526.089,A -85,B 0,C 180,E1 -17920.574,E2 -17920.574} C_VEL
LIN {X 0,Y 268.073,Z 527.46,A -85,B 0,C 180,E1 -17922.108,E2 -17922.108} C_VEL
LIN {X 0,Y 268.053,Z 528.629,A -85,B 0,C 180,E1 -17924.047,E2 -17924.047} C_VEL
LIN {X 0,Y 268.133,Z 529.115,A -85,B 0,C 180,E1 -17926.758,E2 -17926.758} C_VEL
LIN {X 0,Y 268.668,Z 528.24,A -85,B 0,C 180,E1 -17929.658,E2 -17929.658} C_VEL
LIN {X 0,Y 269.11,Z 526.975,A -85,B 0,C 180,E1 -17931.447,E2 -17931.447} C_VEL
LIN {X 0,Y 269.67,Z 525.366,A -85,B 0,C 180,E1 -17933.013,E2 -17933.013} C_VEL
LIN {X 0,Y 270.775,Z 522.081,A -85,B 0,C 180,E1 -17935.358,E2 -17935.358} C_VEL
LIN {X 0,Y 272.139,Z 517.628,A -85,B 0,C 180,E1 -17937.701,E2 -17937.701} C_VEL
LIN {X 0,Y 273.913,Z 511.874,A -85,B 0,C 180,E1 -17940.022,E2 -17940.022} C_VEL
LIN {X 0,Y 276.076,Z 504.562,A -85,B 0,C 180,E1 -17942.317,E2 -17942.317} C_VEL
LIN {X 0,Y 278.126,Z 497.006,A -85,B 0,C 180,E1 -17944.211,E2 -17944.211} C_VEL
LIN {X 0,Y 280.515,Z 487.767,A -85,B 0,C 180,E1 -17946.07,E2 -17946.07} C_VEL
LIN {X 0,Y 282.977,Z 477.254,A -85,B 0,C 180,E1 -17947.753,E2 -17947.753} C_VEL
LIN {X 0,Y 285.151,Z 466,A -85,B 0,C 180,E1 -17949.167,E2 -17949.167} C_VEL
LIN {X 0,Y 286.922,Z 454.861,A -85,B 0,C 180,E1 -17950.259,E2 -17950.259} C_VEL
LIN {X 0,Y 288.413,Z 442.936,A -85,B 0,C 180,E1 -17951.143,E2 -17951.143} C_VEL
LIN {X 0,Y 289.542,Z 429.852,A -85,B 0,C 180,E1 -17951.817,E2 -17951.817} C_VEL
LIN {X 0,Y 290.269,Z 414.671,A -85,B 0,C 180,E1 -17952.272,E2 -17952.272} C_VEL
LIN {X 0,Y 292.351,Z 360.396,A -85,B 0,C 180,E1 -17953.598,E2 -17953.598} C_VEL
LIN {X 0,Y 285.357,Z 345.213,A -85,B 0,C 180,E1 -17955.046,E2 -17955.046} C_VEL
LIN {X 0,Y 277.325,Z 330.356,A -85,B 0,C 180,E1 -17956.762,E2 -17956.762} C_VEL
LIN {X 0,Y 272.532,Z 322.258,A -85,B 0,C 180,E1 -17957.829,E2 -17957.829} C_VEL
LIN {X 0,Y 270.775,Z 318.958,A -85,B 0,C 180,E1 -17958.284,E2 -17958.284} C_VEL
LIN {X 0,Y 270.196,Z 316.825,A -85,B 0,C 180,E1 -17959.268,E2 -17959.268} C_VEL
LIN {X 0,Y 270.22,Z 316.828,A -85,B 0,C 180,E1 -17963.259,E2 -17963.259} C_VEL
LIN {X 0,Y 270.205,Z 316.823,A -85,B 0,C 180,E1 -17966.893,E2 -17966.893} C_VEL
LIN {X 0,Y 270.231,Z 316.817,A -85,B 0,C 180,E1 -17970.387,E2 -17970.387} C_VEL
LIN {X 0,Y 270.266,Z 316.813,A -85,B 0,C 180,E1 -17973.764,E2 -17973.764} C_VEL
LIN {X 0,Y 270.235,Z 316.814,A -85,B 0,C 180,E1 -17977.039,E2 -17977.039} C_VEL
LIN {X 0,Y 270.304,Z 316.808,A -85,B 0,C 180,E1 -17980.244,E2 -17980.244} C_VEL
LIN {X 0,Y 270.405,Z 316.792,A -85,B 0,C 180,E1 -17984.935,E2 -17984.935} C_VEL
LIN {X 0,Y 270.354,Z 316.796,A -85,B 0,C 180,E1 -17985.959,E2 -17985.959} C_VEL
LIN {X 0,Y 269.726,Z 316.883,A -85,B 0,C 180,E1 -17987.203,E2 -17987.203} C_VEL
LIN {X 0,Y 267.025,Z 317.224,A -85,B 0,C 180,E1 -17989.235,E2 -17989.235} C_VEL
LIN {X 0,Y 263.901,Z 317.613,A -85,B 0,C 180,E1 -17991.731,E2 -17991.731} C_VEL
LIN {X 0,Y 263.552,Z 317.652,A -85,B 0,C 180,E1 -17992.593,E2 -17992.593} C_VEL
LIN {X 0,Y 263.752,Z 317.629,A -85,B 0,C 180,E1 -17998.473,E2 -17998.473} C_VEL
LIN {X 0,Y 263.752,Z 317.613,A -85,B 0,C 180,E1 -18001.527,E2 -18001.527} C_VEL
LIN {X 0,Y 263.575,Z 317.644,A -85,B 0,C 180,E1 -18007.661,E2 -18007.661} C_VEL
LIN {X 0,Y 263.376,Z 317.66,A -85,B 0,C 180,E1 -18010.765,E2 -18010.765} C_VEL
LIN {X 0,Y 263.353,Z 317.669,A -85,B 0,C 180,E1 -18015.478,E2 -18015.478} C_VEL
LIN {X 0,Y 263.265,Z 317.682,A -85,B 0,C 180,E1 -18020.306,E2 -18020.306} C_VEL
LIN {X 0,Y 263.194,Z 317.688,A -85,B 0,C 180,E1 -18025.293,E2 -18025.293} C_VEL
LIN {X 0,Y 263.182,Z 317.697,A -85,B 0,C 180,E1 -18028.729,E2 -18028.729} C_VEL
LIN {X 0,Y 263.135,Z 317.707,A -85,B 0,C 180,E1 -18032.288,E2 -18032.288} C_VEL
LIN {X 0,Y 263.185,Z 317.696,A -85,B 0,C 180,E1 -18036.763,E2 -18036.763} C_VEL
LIN {X 0,Y 263.126,Z 317.708,A -85,B 0,C 180,E1 -18041.593,E2 -18041.593} C_VEL
LIN {X 0,Y 263.107,Z 317.708,A -85,B 0,C 180,E1 -18046.155,E2 -18046.155} C_VEL
LIN {X 0,Y 263.145,Z 317.819,A -85,B 0,C 180,E1 -18047.981,E2 -18047.981} C_VEL
LIN {X 0,Y 265.668,Z 326.423,A -85,B 0,C 180,E1 -18051.906,E2 -18051.906} C_VEL
LIN {X 0,Y 267.723,Z 334.525,A -85,B 0,C 180,E1 -18055.283,E2 -18055.283} C_VEL
LIN {X 0,Y 270.01,Z 338.976,A -85,B 0,C 180,E1 -18055.839,E2 -18055.839} C_VEL
LIN {X 0,Y 277.221,Z 353.324,A -85,B 0,C 180,E1 -18057.505,E2 -18057.505} C_VEL
LIN {X 0,Y 281.271,Z 362.424,A -85,B 0,C 180,E1 -18058.42,E2 -18058.42} C_VEL
LIN {X 0,Y 284.977,Z 383.211,A -85,B 0,C 180,E1 -18059.602,E2 -18059.602} C_VEL
LIN {X 0,Y 285.576,Z 388.72,A -85,B 0,C 180,E1 -18059.855,E2 -18059.855} C_VEL
LIN {X 0,Y 283.314,Z 444.68,A -85,B 0,C 180,E1 -18061.293,E2 -18061.293} C_VEL
LIN {X 0,Y 281.935,Z 458.762,A -85,B 0,C 180,E1 -18061.932,E2 -18061.932} C_VEL
LIN {X 0,Y 280.22,Z 470.915,A -85,B 0,C 180,E1 -18062.76,E2 -18062.76} C_VEL
LIN {X 0,Y 277.891,Z 483.441,A -85,B 0,C 180,E1 -18063.932,E2 -18063.932} C_VEL
LIN {X 0,Y 275.58,Z 494.605,A -85,B 0,C 180,E1 -18065.316,E2 -18065.316} C_VEL
LIN {X 0,Y 272.999,Z 504.716,A -85,B 0,C 180,E1 -18066.883,E2 -18066.883} C_VEL
LIN {X 0,Y 270.505,Z 513.836,A -85,B 0,C 180,E1 -18068.669,E2 -18068.669} C_VEL
LIN {X 0,Y 268.182,Z 521.917,A -85,B 0,C 180,E1 -18070.634,E2 -18070.634} C_VEL
LIN {X 0,Y 265.971,Z 529.942,A -85,B 0,C 180,E1 -18073.101,E2 -18073.101} C_VEL
LIN {X 0,Y 264.167,Z 535.73,A -85,B 0,C 180,E1 -18075.359,E2 -18075.359} C_VEL
LIN {X 0,Y 262.813,Z 540.312,A -85,B 0,C 180,E1 -18077.646,E2 -18077.646} C_VEL
LIN {X 0,Y 261.952,Z 543.822,A -85,B 0,C 180,E1 -18079.956,E2 -18079.956} C_VEL
LIN {X 0,Y 261.356,Z 546.346,A -85,B 0,C 180,E1 -18082.272,E2 -18082.272} C_VEL
LIN {X 0,Y 261.124,Z 548.047,A -85,B 0,C 180,E1 -18084.769,E2 -18084.769} C_VEL
LIN {X 0,Y 261.106,Z 548.669,A -85,B 0,C 180,E1 -18086.913,E2 -18086.913} C_VEL
LIN {X 0,Y 261.141,Z 548.662,A -85,B 0,C 180,E1 -18088.457,E2 -18088.457} C_VEL
LIN {X 0,Y 261.176,Z 548.261,A -85,B 0,C 180,E1 -18089.999,E2 -18089.999} C_VEL
LIN {X 0,Y 261.164,Z 547.418,A -85,B 0,C 180,E1 -18091.541,E2 -18091.541} C_VEL
LIN {X 0,Y 261.147,Z 546.165,A -85,B 0,C 180,E1 -18093.084,E2 -18093.084} C_VEL
LIN {X 0,Y 261.156,Z 543.617,A -85,B 0,C 180,E1 -18095.307,E2 -18095.307} C_VEL
LIN {X 0,Y 261.362,Z 539.76,A -85,B 0,C 180,E1 -18097.726,E2 -18097.726} C_VEL
LIN {X 0,Y 261.762,Z 534.889,A -85,B 0,C 180,E1 -18100.049,E2 -18100.049} C_VEL
LIN {X 0,Y 262.456,Z 528.724,A -85,B 0,C 180,E1 -18102.369,E2 -18102.369} C_VEL
LIN {X 0,Y 263.647,Z 521.058,A -85,B 0,C 180,E1 -18104.668,E2 -18104.668} C_VEL
LIN {X 0,Y 264.873,Z 513.194,A -85,B 0,C 180,E1 -18106.571,E2 -18106.571} C_VEL
LIN {X 0,Y 266.175,Z 503.539,A -85,B 0,C 180,E1 -18108.471,E2 -18108.471} C_VEL
LIN {X 0,Y 267.634,Z 492.823,A -85,B 0,C 180,E1 -18110.16,E2 -18110.16} C_VEL
LIN {X 0,Y 269.306,Z 480.833,A -85,B 0,C 180,E1 -18111.629,E2 -18111.629} C_VEL
LIN {X 0,Y 270.736,Z 467.939,A -85,B 0,C 180,E1 -18112.814,E2 -18112.814} C_VEL
LIN {X 0,Y 271.925,Z 454.963,A -85,B 0,C 180,E1 -18113.665,E2 -18113.665} C_VEL
LIN {X 0,Y 272.625,Z 442.092,A -85,B 0,C 180,E1 -18114.206,E2 -18114.206} C_VEL
LIN {X 0,Y 274.026,Z 382.785,A -85,B 0,C 180,E1 -18115.762,E2 -18115.762} C_VEL
LIN {X 0,Y 269.206,Z 345.293,A -85,B 0,C 180,E1 -18117.217,E2 -18117.217} C_VEL
LIN {X 0,Y 268.242,Z 339.949,A -85,B 0,C 180,E1 -18117.453,E2 -18117.453} C_VEL
LIN {X 0,Y 266.972,Z 335.933,A -85,B 0,C 180,E1 -18117.702,E2 -18117.702} C_VEL
LIN {X 0,Y 264.893,Z 325.731,A -85,B 0,C 180,E1 -18121.131,E2 -18121.131} C_VEL
LIN {X 0,Y 263.17,Z 317.705,A -85,B 0,C 180,E1 -18123.98,E2 -18123.98} C_VEL
LIN {X 0,Y 263.156,Z 317.704,A -85,B 0,C 180,E1 -18127.896,E2 -18127.896} C_VEL
LIN {X 0,Y 263.119,Z 317.708,A -85,B 0,C 180,E1 -18131.892,E2 -18131.892} C_VEL
LIN {X 0,Y 263.12,Z 317.71,A -85,B 0,C 180,E1 -18136.149,E2 -18136.149} C_VEL
LIN {X 0,Y 263.115,Z 317.706,A -85,B 0,C 180,E1 -18140.129,E2 -18140.129} C_VEL
LIN {X 0,Y 263.182,Z 317.699,A -85,B 0,C 180,E1 -18144.021,E2 -18144.021} C_VEL
LIN {X 0,Y 263.128,Z 317.704,A -85,B 0,C 180,E1 -18147.711,E2 -18147.711} C_VEL
LIN {X 0,Y 263.195,Z 317.697,A -85,B 0,C 180,E1 -18151.782,E2 -18151.782} C_VEL
LIN {X 0,Y 263.219,Z 317.696,A -85,B 0,C 180,E1 -18155.2,E2 -18155.2} C_VEL
LIN {X 0,Y 263.256,Z 317.688,A -85,B 0,C 180,E1 -18159.693,E2 -18159.693} C_VEL
LIN {X 0,Y 263.337,Z 317.673,A -85,B 0,C 180,E1 -18164.521,E2 -18164.521} C_VEL
LIN {X 0,Y 263.366,Z 317.68,A -85,B 0,C 180,E1 -18169.234,E2 -18169.234} C_VEL
LIN {X 0,Y 263.564,Z 317.643,A -85,B 0,C 180,E1 -18172.338,E2 -18172.338} C_VEL
LIN {X 0,Y 263.743,Z 317.628,A -85,B 0,C 180,E1 -18178.473,E2 -18178.473} C_VEL
LIN {X 0,Y 263.743,Z 317.632,A -85,B 0,C 180,E1 -18181.527,E2 -18181.527} C_VEL
LIN {X 0,Y 263.524,Z 317.646,A -85,B 0,C 180,E1 -18187.663,E2 -18187.663} C_VEL
LIN {X 0,Y 263.347,Z 317.678,A -85,B 0,C 180,E1 -18190.767,E2 -18190.767} C_VEL
LIN {X 0,Y 263.343,Z 317.677,A -85,B 0,C 180,E1 -18195.479,E2 -18195.479} C_VEL
LIN {X 0,Y 263.256,Z 317.692,A -85,B 0,C 180,E1 -18200.307,E2 -18200.307} C_VEL
LIN {X 0,Y 263.186,Z 317.698,A -85,B 0,C 180,E1 -18205.294,E2 -18205.294} C_VEL
LIN {X 0,Y 263.173,Z 317.701,A -85,B 0,C 180,E1 -18208.73,E2 -18208.73} C_VEL
LIN {X 0,Y 263.127,Z 317.708,A -85,B 0,C 180,E1 -18212.289,E2 -18212.289} C_VEL
LIN {X 0,Y 263.174,Z 317.703,A -85,B 0,C 180,E1 -18216.763,E2 -18216.763} C_VEL
LIN {X 0,Y 263.086,Z 317.708,A -85,B 0,C 180,E1 -18219.876,E2 -18219.876} C_VEL
LIN {X 0,Y 263.071,Z 317.71,A -85,B 0,C 180,E1 -18223.995,E2 -18223.995} C_VEL
LIN {X 0,Y 263.076,Z 317.712,A -85,B 0,C 180,E1 -18228.419,E2 -18228.419} C_VEL
LIN {X 0,Y 263.154,Z 317.702,A -85,B 0,C 180,E1 -18232.104,E2 -18232.104} C_VEL
LIN {X 0,Y 263.148,Z 317.704,A -85,B 0,C 180,E1 -18235.887,E2 -18235.887} C_VEL
LIN {X 0,Y 263.123,Z 317.708,A -85,B 0,C 180,E1 -18239.505,E2 -18239.505} C_VEL
LIN {X 0,Y 263.139,Z 317.707,A -85,B 0,C 180,E1 -18242.998,E2 -18242.998} C_VEL
LIN {X 0,Y 263.143,Z 317.705,A -85,B 0,C 180,E1 -18246.385,E2 -18246.385} C_VEL
LIN {X 0,Y 263.237,Z 317.695,A -85,B 0,C 180,E1 -18249.693,E2 -18249.693} C_VEL
LIN {X 0,Y 263.315,Z 317.685,A -85,B 0,C 180,E1 -18254.521,E2 -18254.521} C_VEL
LIN {X 0,Y 263.357,Z 317.796,A -85,B 0,C 180,E1 -18255.907,E2 -18255.907} C_VEL
LIN {X 0,Y 263.49,Z 318.396,A -85,B 0,C 180,E1 -18256.087,E2 -18256.087} C_VEL
LIN {X 0,Y 272.049,Z 341.215,A -85,B 0,C 180,E1 -18257.508,E2 -18257.508} C_VEL
LIN {X 0,Y 274.368,Z 349.08,A -85,B 0,C 180,E1 -18257.924,E2 -18257.924} C_VEL
LIN {X 0,Y 274.97,Z 352.3,A -85,B 0,C 180,E1 -18258.064,E2 -18258.064} C_VEL
LIN {X 0,Y 272.815,Z 424.879,A -85,B 0,C 180,E1 -18259.94,E2 -18259.94} C_VEL
LIN {X 0,Y 272.115,Z 437.548,A -85,B 0,C 180,E1 -18260.524,E2 -18260.524} C_VEL
LIN {X 0,Y 271.087,Z 450.533,A -85,B 0,C 180,E1 -18261.428,E2 -18261.428} C_VEL
LIN {X 0,Y 269.986,Z 462.025,A -85,B 0,C 180,E1 -18262.523,E2 -18262.523} C_VEL
LIN {X 0,Y 268.609,Z 473.808,A -85,B 0,C 180,E1 -18263.994,E2 -18263.994} C_VEL
LIN {X 0,Y 267.082,Z 484.391,A -85,B 0,C 180,E1 -18265.662,E2 -18265.662} C_VEL
LIN {X 0,Y 265.736,Z 493.042,A -85,B 0,C 180,E1 -18267.348,E2 -18267.348} C_VEL
LIN {X 0,Y 264.502,Z 501.001,A -85,B 0,C 180,E1 -18269.24,E2 -18269.24} C_VEL
LIN {X 0,Y 263.28,Z 508.788,A -85,B 0,C 180,E1 -18271.531,E2 -18271.531} C_VEL
LIN {X 0,Y 262.394,Z 515.019,A -85,B 0,C 180,E1 -18273.84,E2 -18273.84} C_VEL
LIN {X 0,Y 261.737,Z 520.652,A -85,B 0,C 180,E1 -18276.533,E2 -18276.533} C_VEL
LIN {X 0,Y 261.192,Z 524.868,A -85,B 0,C 180,E1 -18279.292,E2 -18279.292} C_VEL
LIN {X 0,Y 261.003,Z 526.599,A -85,B 0,C 180,E1 -18280.866,E2 -18280.866} C_VEL
LIN {X 0,Y 260.962,Z 527.917,A -85,B 0,C 180,E1 -18282.443,E2 -18282.443} C_VEL
LIN {X 0,Y 260.97,Z 528.899,A -85,B 0,C 180,E1 -18284.188,E2 -18284.188} C_VEL
LIN {X 0,Y 261.098,Z 529.36,A -85,B 0,C 180,E1 -18287.224,E2 -18287.224} C_VEL
LIN {X 0,Y 261.616,Z 528.524,A -85,B 0,C 180,E1 -18289.908,E2 -18289.908} C_VEL
LIN {X 0,Y 262.202,Z 527,A -85,B 0,C 180,E1 -18292.041,E2 -18292.041} C_VEL
LIN {X 0,Y 263.421,Z 523.716,A -85,B 0,C 180,E1 -18294.89,E2 -18294.89} C_VEL
LIN {X 0,Y 265.006,Z 519.015,A -85,B 0,C 180,E1 -18297.653,E2 -18297.653} C_VEL
LIN {X 0,Y 266.797,Z 513.545,A -85,B 0,C 180,E1 -18300.034,E2 -18300.034} C_VEL
LIN {X 0,Y 268.964,Z 506.607,A -85,B 0,C 180,E1 -18302.39,E2 -18302.39} C_VEL
LIN {X 0,Y 271.144,Z 499.106,A -85,B 0,C 180,E1 -18304.419,E2 -18304.419} C_VEL
LIN {X 0,Y 273.751,Z 489.777,A -85,B 0,C 180,E1 -18306.42,E2 -18306.42} C_VEL
LIN {X 0,Y 276.403,Z 479.156,A -85,B 0,C 180,E1 -18308.21,E2 -18308.21} C_VEL
LIN {X 0,Y 278.821,Z 467.461,A -85,B 0,C 180,E1 -18309.763,E2 -18309.763} C_VEL
LIN {X 0,Y 280.686,Z 456.283,A -85,B 0,C 180,E1 -18310.908,E2 -18310.908} C_VEL
LIN {X 0,Y 282.319,Z 444.113,A -85,B 0,C 180,E1 -18311.845,E2 -18311.845} C_VEL
LIN {X 0,Y 283.496,Z 431.372,A -85,B 0,C 180,E1 -18312.543,E2 -18312.543} C_VEL
LIN {X 0,Y 284.221,Z 417.636,A -85,B 0,C 180,E1 -18312.99,E2 -18312.99} C_VEL
LIN {X 0,Y 286.454,Z 362.471,A -85,B 0,C 180,E1 -18314.357,E2 -18314.357} C_VEL
LIN {X 0,Y 280.064,Z 348.609,A -85,B 0,C 180,E1 -18315.738,E2 -18315.738} C_VEL
LIN {X 0,Y 271.108,Z 331.874,A -85,B 0,C 180,E1 -18317.748,E2 -18317.748} C_VEL
LIN {X 0,Y 265.482,Z 322.787,A -85,B 0,C 180,E1 -18319.065,E2 -18319.065} C_VEL
LIN {X 0,Y 263.54,Z 319.346,A -85,B 0,C 180,E1 -18319.582,E2 -18319.582} C_VEL
LIN {X 0,Y 263.129,Z 317.694,A -85,B 0,C 180,E1 -18320.419,E2 -18320.419} C_VEL
LIN {X 0,Y 263.166,Z 317.702,A -85,B 0,C 180,E1 -18324.018,E2 -18324.018} C_VEL
LIN {X 0,Y 263.136,Z 317.705,A -85,B 0,C 180,E1 -18327.712,E2 -18327.712} C_VEL
LIN {X 0,Y 263.204,Z 317.699,A -85,B 0,C 180,E1 -18331.783,E2 -18331.783} C_VEL
LIN {X 0,Y 263.229,Z 317.697,A -85,B 0,C 180,E1 -18335.2,E2 -18335.2} C_VEL
LIN {X 0,Y 263.266,Z 317.688,A -85,B 0,C 180,E1 -18339.693,E2 -18339.693} C_VEL
LIN {X 0,Y 263.353,Z 317.674,A -85,B 0,C 180,E1 -18344.522,E2 -18344.522} C_VEL
LIN {X 0,Y 263.376,Z 317.67,A -85,B 0,C 180,E1 -18349.234,E2 -18349.234} C_VEL
LIN {X 0,Y 263.575,Z 317.652,A -85,B 0,C 180,E1 -18352.338,E2 -18352.338} C_VEL
LIN {X 0,Y 263.552,Z 317.652,A -85,B 0,C 180,E1 -18352.593,E2 -18352.593} C_VEL
LIN {X 0,Y 262.836,Z 317.742,A -85,B 0,C 180,E1 -18353.868,E2 -18353.868} C_VEL
LIN {X 0,Y 260.041,Z 318.087,A -85,B 0,C 180,E1 -18355.949,E2 -18355.949} C_VEL
LIN {X 0,Y 257.732,Z 318.377,A -85,B 0,C 180,E1 -18357.642,E2 -18357.642} C_VEL
LIN {X 0,Y 256.78,Z 318.496,A -85,B 0,C 180,E1 -18358.952,E2 -18358.952} C_VEL
LIN {X 0,Y 256.719,Z 318.494,A -85,B 0,C 180,E1 -18359.395,E2 -18359.395} C_VEL
LIN {X 0,Y 256.715,Z 318.49,A -85,B 0,C 180,E1 -18361.569,E2 -18361.569} C_VEL
LIN {X 0,Y 256.542,Z 318.522,A -85,B 0,C 180,E1 -18367.873,E2 -18367.873} C_VEL
LIN {X 0,Y 256.312,Z 318.539,A -85,B 0,C 180,E1 -18371.066,E2 -18371.066} C_VEL
LIN {X 0,Y 256.302,Z 318.544,A -85,B 0,C 180,E1 -18375.915,E2 -18375.915} C_VEL
LIN {X 0,Y 256.165,Z 318.563,A -85,B 0,C 180,E1 -18380.895,E2 -18380.895} C_VEL
LIN {X 0,Y 256.173,Z 318.563,A -85,B 0,C 180,E1 -18385.13,E2 -18385.13} C_VEL
LIN {X 0,Y 256.116,Z 318.57,A -85,B 0,C 180,E1 -18389.599,E2 -18389.599} C_VEL
LIN {X 0,Y 256.07,Z 318.578,A -85,B 0,C 180,E1 -18393.292,E2 -18393.292} C_VEL
LIN {X 0,Y 256.117,Z 318.574,A -85,B 0,C 180,E1 -18397.27,E2 -18397.27} C_VEL
LIN {X 0,Y 256.056,Z 318.585,A -85,B 0,C 180,E1 -18401.203,E2 -18401.203} C_VEL
LIN {X 0,Y 256.043,Z 318.588,A -85,B 0,C 180,E1 -18405.534,E2 -18405.534} C_VEL
LIN {X 0,Y 256.108,Z 318.642,A -85,B 0,C 180,E1 -18406.765,E2 -18406.765} C_VEL
LIN {X 0,Y 258.586,Z 327.347,A -85,B 0,C 180,E1 -18410.922,E2 -18410.922} C_VEL
LIN {X 0,Y 260.534,Z 334.392,A -85,B 0,C 180,E1 -18413.953,E2 -18413.953} C_VEL
LIN {X 0,Y 268.935,Z 350.408,A -85,B 0,C 180,E1 -18416.044,E2 -18416.044} C_VEL
LIN {X 0,Y 275.631,Z 364.745,A -85,B 0,C 180,E1 -18417.625,E2 -18417.625} C_VEL
LIN {X 0,Y 278.935,Z 382.735,A -85,B 0,C 180,E1 -18418.711,E2 -18418.711} C_VEL
LIN {X 0,Y 279.773,Z 389.17,A -85,B 0,C 180,E1 -18419.037,E2 -18419.037} C_VEL
LIN {X 0,Y 277.462,Z 443.805,A -85,B 0,C 180,E1 -18420.455,E2 -18420.455} C_VEL
LIN {X 0,Y 276.146,Z 457.574,A -85,B 0,C 180,E1 -18421.081,E2 -18421.081} C_VEL
LIN {X 0,Y 274.342,Z 470.009,A -85,B 0,C 180,E1 -18421.918,E2 -18421.918} C_VEL
LIN {X 0,Y 272.256,Z 481.127,A -85,B 0,C 180,E1 -18422.936,E2 -18422.936} C_VEL
LIN {X 0,Y 270.007,Z 491.393,A -85,B 0,C 180,E1 -18424.151,E2 -18424.151} C_VEL
LIN {X 0,Y 267.375,Z 502.024,A -85,B 0,C 180,E1 -18425.75,E2 -18425.75} C_VEL
LIN {X 0,Y 264.895,Z 510.74,A -85,B 0,C 180,E1 -18427.374,E2 -18427.374} C_VEL
LIN {X 0,Y 262.513,Z 518.777,A -85,B 0,C 180,E1 -18429.222,E2 -18429.222} C_VEL
LIN {X 0,Y 260.171,Z 526.693,A -85,B 0,C 180,E1 -18431.493,E2 -18431.493} C_VEL
LIN {X 0,Y 258.548,Z 532.07,A -85,B 0,C 180,E1 -18433.415,E2 -18433.415} C_VEL
LIN {X 0,Y 256.727,Z 537.366,A -85,B 0,C 180,E1 -18435.736,E2 -18435.736} C_VEL
LIN {X 0,Y 255.507,Z 541.513,A -85,B 0,C 180,E1 -18438.094,E2 -18438.094} C_VEL
LIN {X 0,Y 254.683,Z 544.63,A -85,B 0,C 180,E1 -18440.469,E2 -18440.469} C_VEL
LIN {X 0,Y 254.314,Z 546.2,A -85,B 0,C 180,E1 -18442.057,E2 -18442.057} C_VEL
LIN {X 0,Y 254.014,Z 548.066,A -85,B 0,C 180,E1 -18445.238,E2 -18445.238} C_VEL
LIN {X 0,Y 254.02,Z 548.417,A -85,B 0,C 180,E1 -18446.827,E2 -18446.827} C_VEL
LIN {X 0,Y 254.068,Z 548.384,A -85,B 0,C 180,E1 -18448.414,E2 -18448.414} C_VEL
LIN {X 0,Y 254.101,Z 547.937,A -85,B 0,C 180,E1 -18449.999,E2 -18449.999} C_VEL
LIN {X 0,Y 254.091,Z 547.06,A -85,B 0,C 180,E1 -18451.584,E2 -18451.584} C_VEL
LIN {X 0,Y 254.06,Z 545.779,A -85,B 0,C 180,E1 -18453.17,E2 -18453.17} C_VEL
LIN {X 0,Y 254.053,Z 543.523,A -85,B 0,C 180,E1 -18455.196,E2 -18455.196} C_VEL
LIN {X 0,Y 254.313,Z 539.255,A -85,B 0,C 180,E1 -18457.941,E2 -18457.941} C_VEL
LIN {X 0,Y 254.734,Z 534.318,A -85,B 0,C 180,E1 -18460.33,E2 -18460.33} C_VEL
LIN {X 0,Y 255.488,Z 528.083,A -85,B 0,C 180,E1 -18462.711,E2 -18462.711} C_VEL
LIN {X 0,Y 256.712,Z 520.309,A -85,B 0,C 180,E1 -18465.073,E2 -18465.073} C_VEL
LIN {X 0,Y 257.977,Z 512.325,A -85,B 0,C 180,E1 -18467.028,E2 -18467.028} C_VEL
LIN {X 0,Y 259.428,Z 502.555,A -85,B 0,C 180,E1 -18468.969,E2 -18468.969} C_VEL
LIN {X 0,Y 260.737,Z 492.992,A -85,B 0,C 180,E1 -18470.511,E2 -18470.511} C_VEL
LIN {X 0,Y 262.228,Z 482.768,A -85,B 0,C 180,E1 -18471.829,E2 -18471.829} C_VEL
LIN {X 0,Y 263.718,Z 470.711,A -85,B 0,C 180,E1 -18473.041,E2 -18473.041} C_VEL
LIN {X 0,Y 264.914,Z 458.034,A -85,B 0,C 180,E1 -18473.967,E2 -18473.967} C_VEL
LIN {X 0,Y 265.807,Z 444.948,A -85,B 0,C 180,E1 -18474.608,E2 -18474.608} C_VEL
LIN {X 0,Y 267.439,Z 383.982,A -85,B 0,C 180,E1 -18476.264,E2 -18476.264} C_VEL
LIN {X 0,Y 262.457,Z 344.748,A -85,B 0,C 180,E1 -18477.831,E2 -18477.831} C_VEL
LIN {X 0,Y 261.401,Z 340.691,A -85,B 0,C 180,E1 -18478.047,E2 -18478.047} C_VEL
LIN {X 0,Y 259.715,Z 335.616,A -85,B 0,C 180,E1 -18478.386,E2 -18478.386} C_VEL
LIN {X 0,Y 257.6,Z 325.473,A -85,B 0,C 180,E1 -18481.921,E2 -18481.921} C_VEL
LIN {X 0,Y 256.118,Z 318.582,A -85,B 0,C 180,E1 -18484.449,E2 -18484.449} C_VEL
LIN {X 0,Y 256.112,Z 318.58,A -85,B 0,C 180,E1 -18487.27,E2 -18487.27} C_VEL
LIN {X 0,Y 256.05,Z 318.587,A -85,B 0,C 180,E1 -18491.202,E2 -18491.202} C_VEL
LIN {X 0,Y 256.05,Z 318.589,A -85,B 0,C 180,E1 -18495.53,E2 -18495.53} C_VEL
LIN {X 0,Y 256.057,Z 318.587,A -85,B 0,C 180,E1 -18498.797,E2 -18498.797} C_VEL
LIN {X 0,Y 256.139,Z 318.58,A -85,B 0,C 180,E1 -18502.869,E2 -18502.869} C_VEL
LIN {X 0,Y 256.079,Z 318.587,A -85,B 0,C 180,E1 -18506.709,E2 -18506.709} C_VEL
LIN {X 0,Y 256.132,Z 318.577,A -85,B 0,C 180,E1 -18511.404,E2 -18511.404} C_VEL
LIN {X 0,Y 256.16,Z 318.573,A -85,B 0,C 180,E1 -18515.698,E2 -18515.698} C_VEL
LIN {X 0,Y 256.16,Z 318.576,A -85,B 0,C 180,E1 -18519.104,E2 -18519.104} C_VEL
LIN {X 0,Y 256.287,Z 318.551,A -85,B 0,C 180,E1 -18524.084,E2 -18524.084} C_VEL
LIN {X 0,Y 256.302,Z 318.558,A -85,B 0,C 180,E1 -18528.934,E2 -18528.934} C_VEL
LIN {X 0,Y 256.532,Z 318.519,A -85,B 0,C 180,E1 -18532.127,E2 -18532.127} C_VEL
LIN {X 0,Y 256.706,Z 318.505,A -85,B 0,C 180,E1 -18538.431,E2 -18538.431} C_VEL
LIN {X 0,Y 256.706,Z 318.508,A -85,B 0,C 180,E1 -18541.569,E2 -18541.569} C_VEL
LIN {X 0,Y 256.447,Z 318.523,A -85,B 0,C 180,E1 -18546.587,E2 -18546.587} C_VEL
LIN {X 0,Y 256.419,Z 318.537,A -85,B 0,C 180,E1 -18549.465,E2 -18549.465} C_VEL
LIN {X 0,Y 256.248,Z 318.562,A -85,B 0,C 180,E1 -18554.291,E2 -18554.291} C_VEL
LIN {X 0,Y 256.204,Z 318.568,A -85,B 0,C 180,E1 -18557.563,E2 -18557.563} C_VEL
LIN {X 0,Y 256.146,Z 318.573,A -85,B 0,C 180,E1 -18561.118,E2 -18561.118} C_VEL
LIN {X 0,Y 256.164,Z 318.573,A -85,B 0,C 180,E1 -18565.131,E2 -18565.131} C_VEL
LIN {X 0,Y 256.108,Z 318.579,A -85,B 0,C 180,E1 -18569.601,E2 -18569.601} C_VEL
LIN {X 0,Y 256.062,Z 318.582,A -85,B 0,C 180,E1 -18573.294,E2 -18573.294} C_VEL
LIN {X 0,Y 256.107,Z 318.58,A -85,B 0,C 180,E1 -18577.271,E2 -18577.271} C_VEL
LIN {X 0,Y 256.013,Z 318.593,A -85,B 0,C 180,E1 -18581.212,E2 -18581.212} C_VEL
LIN {X 0,Y 256.013,Z 318.592,A -85,B 0,C 180,E1 -18585.541,E2 -18585.541} C_VEL
LIN {X 0,Y 256.014,Z 318.593,A -85,B 0,C 180,E1 -18588.791,E2 -18588.791} C_VEL
LIN {X 0,Y 256.124,Z 318.58,A -85,B 0,C 180,E1 -18592.868,E2 -18592.868} C_VEL
LIN {X 0,Y 256.063,Z 318.587,A -85,B 0,C 180,E1 -18596.708,E2 -18596.708} C_VEL
LIN {X 0,Y 256.052,Z 318.586,A -85,B 0,C 180,E1 -18600.394,E2 -18600.394} C_VEL
LIN {X 0,Y 256.131,Z 318.58,A -85,B 0,C 180,E1 -18604.89,E2 -18604.89} C_VEL
LIN {X 0,Y 256.146,Z 318.574,A -85,B 0,C 180,E1 -18609.105,E2 -18609.105} C_VEL
LIN {X 0,Y 256.249,Z 318.564,A -85,B 0,C 180,E1 -18614.083,E2 -18614.083} C_VEL
LIN {X 0,Y 256.317,Z 318.559,A -85,B 0,C 180,E1 -18615.359,E2 -18615.359} C_VEL
LIN {X 0,Y 257.42,Z 321.599,A -85,B 0,C 180,E1 -18615.602,E2 -18615.602} C_VEL
LIN {X 0,Y 264.991,Z 341.357,A -85,B 0,C 180,E1 -18616.897,E2 -18616.897} C_VEL
LIN {X 0,Y 267.938,Z 350.908,A -85,B 0,C 180,E1 -18617.432,E2 -18617.432} C_VEL
LIN {X 0,Y 268.364,Z 353.857,A -85,B 0,C 180,E1 -18617.553,E2 -18617.553} C_VEL
LIN {X 0,Y 266.106,Z 425.422,A -85,B 0,C 180,E1 -18619.444,E2 -18619.444} C_VEL
LIN {X 0,Y 265.353,Z 438.722,A -85,B 0,C 180,E1 -18620.088,E2 -18620.088} C_VEL
LIN {X 0,Y 264.281,Z 451.482,A -85,B 0,C 180,E1 -18621.013,E2 -18621.013} C_VEL
LIN {X 0,Y 263.15,Z 462.803,A -85,B 0,C 180,E1 -18622.134,E2 -18622.134} C_VEL
LIN {X 0,Y 261.718,Z 474.543,A -85,B 0,C 180,E1 -18623.653,E2 -18623.653} C_VEL
LIN {X 0,Y 260.148,Z 484.982,A -85,B 0,C 180,E1 -18625.352,E2 -18625.352} C_VEL
LIN {X 0,Y 258.614,Z 494.457,A -85,B 0,C 180,E1 -18627.275,E2 -18627.275} C_VEL
LIN {X 0,Y 257.147,Z 503.563,A -85,B 0,C 180,E1 -18629.61,E2 -18629.61} C_VEL
LIN {X 0,Y 255.986,Z 510.908,A -85,B 0,C 180,E1 -18631.968,E2 -18631.968} C_VEL
LIN {X 0,Y 255.248,Z 515.881,A -85,B 0,C 180,E1 -18633.948,E2 -18633.948} C_VEL
LIN {X 0,Y 254.646,Z 520.997,A -85,B 0,C 180,E1 -18636.5,E2 -18636.5} C_VEL
LIN {X 0,Y 254.205,Z 524.421,A -85,B 0,C 180,E1 -18638.747,E2 -18638.747} C_VEL
LIN {X 0,Y 253.883,Z 527.11,A -85,B 0,C 180,E1 -18641.174,E2 -18641.174} C_VEL
LIN {X 0,Y 253.851,Z 528.375,A -85,B 0,C 180,E1 -18642.797,E2 -18642.797} C_VEL
LIN {X 0,Y 253.876,Z 529.198,A -85,B 0,C 180,E1 -18644.428,E2 -18644.428} C_VEL
LIN {X 0,Y 253.882,Z 529.602,A -85,B 0,C 180,E1 -18646.072,E2 -18646.072} C_VEL
LIN {X 0,Y 254.072,Z 529.604,A -85,B 0,C 180,E1 -18647.716,E2 -18647.716} C_VEL
LIN {X 0,Y 254.603,Z 528.797,A -85,B 0,C 180,E1 -18650.193,E2 -18650.193} C_VEL
LIN {X 0,Y 255.332,Z 527.027,A -85,B 0,C 180,E1 -18652.666,E2 -18652.666} C_VEL
LIN {X 0,Y 256.523,Z 524.02,A -85,B 0,C 180,E1 -18655.296,E2 -18655.296} C_VEL
LIN {X 0,Y 257.859,Z 520.32,A -85,B 0,C 180,E1 -18657.604,E2 -18657.604} C_VEL
LIN {X 0,Y 259.889,Z 514.55,A -85,B 0,C 180,E1 -18660.311,E2 -18660.311} C_VEL
LIN {X 0,Y 262.274,Z 507.333,A -85,B 0,C 180,E1 -18662.864,E2 -18662.864} C_VEL
LIN {X 0,Y 264.909,Z 498.801,A -85,B 0,C 180,E1 -18665.221,E2 -18665.221} C_VEL
LIN {X 0,Y 267.517,Z 489.757,A -85,B 0,C 180,E1 -18667.175,E2 -18667.175} C_VEL
LIN {X 0,Y 270.106,Z 479.824,A -85,B 0,C 180,E1 -18668.883,E2 -18668.883} C_VEL
LIN {X 0,Y 272.506,Z 468.848,A -85,B 0,C 180,E1 -18670.39,E2 -18670.39} C_VEL
LIN {X 0,Y 274.705,Z 456.44,A -85,B 0,C 180,E1 -18671.697,E2 -18671.697} C_VEL
LIN {X 0,Y 276.419,Z 443.989,A -85,B 0,C 180,E1 -18672.668,E2 -18672.668} C_VEL
LIN {X 0,Y 277.646,Z 431.147,A -85,B 0,C 180,E1 -18673.37,E2 -18673.37} C_VEL
LIN {X 0,Y 278.484,Z 415.94,A -85,B 0,C 180,E1 -18673.847,E2 -18673.847} C_VEL
LIN {X 0,Y 280.627,Z 364.654,A -85,B 0,C 180,E1 -18675.142,E2 -18675.142} C_VEL
LIN {X 0,Y 274.703,Z 351.708,A -85,B 0,C 180,E1 -18676.487,E2 -18676.487} C_VEL
LIN {X 0,Y 265.969,Z 335.52,A -85,B 0,C 180,E1 -18678.528,E2 -18678.528} C_VEL
LIN {X 0,Y 260.803,Z 327.085,A -85,B 0,C 180,E1 -18679.797,E2 -18679.797} C_VEL
LIN {X 0,Y 258.561,Z 323.489,A -85,B 0,C 180,E1 -18680.371,E2 -18680.371} C_VEL
LIN {X 0,Y 256.449,Z 320.089,A -85,B 0,C 180,E1 -18680.926,E2 -18680.926} C_VEL
LIN {X 0,Y 256.241,Z 319.418,A -85,B 0,C 180,E1 -18681.141,E2 -18681.141} C_VEL
LIN {X 0,Y 256.101,Z 318.572,A -85,B 0,C 180,E1 -18681.617,E2 -18681.617} C_VEL
LIN {X 0,Y 256.108,Z 318.586,A -85,B 0,C 180,E1 -18685.412,E2 -18685.412} C_VEL
LIN {X 0,Y 256.095,Z 318.587,A -85,B 0,C 180,E1 -18688.572,E2 -18688.572} C_VEL
LIN {X 0,Y 256.145,Z 318.576,A -85,B 0,C 180,E1 -18692.196,E2 -18692.196} C_VEL
LIN {X 0,Y 256.17,Z 318.573,A -85,B 0,C 180,E1 -18695.699,E2 -18695.699} C_VEL
LIN {X 0,Y 256.17,Z 318.576,A -85,B 0,C 180,E1 -18699.105,E2 -18699.105} C_VEL
LIN {X 0,Y 256.303,Z 318.555,A -85,B 0,C 180,E1 -18704.085,E2 -18704.085} C_VEL
LIN {X 0,Y 256.312,Z 318.554,A -85,B 0,C 180,E1 -18708.934,E2 -18708.934} C_VEL
LIN {X 0,Y 256.542,Z 318.524,A -85,B 0,C 180,E1 -18712.127,E2 -18712.127} C_VEL
LIN {X 0,Y 256.715,Z 318.506,A -85,B 0,C 180,E1 -18718.431,E2 -18718.431} C_VEL
LIN {X 0,Y 256.719,Z 318.494,A -85,B 0,C 180,E1 -18719.395,E2 -18719.395} C_VEL
LIN {X 0,Y 256.038,Z 318.578,A -85,B 0,C 180,E1 -18720.702,E2 -18720.702} C_VEL
LIN {X 0,Y 252.992,Z 318.967,A -85,B 0,C 180,E1 -18722.824,E2 -18722.824} C_VEL
LIN {X 0,Y 250.456,Z 319.279,A -85,B 0,C 180,E1 -18724.555,E2 -18724.555} C_VEL
LIN {X 0,Y 249.469,Z 319.392,A -85,B 0,C 180,E1 -18725.902,E2 -18725.902} C_VEL
LIN {X 0,Y 249.445,Z 319.395,A -85,B 0,C 180,E1 -18726.358,E2 -18726.358} C_VEL
LIN {X 0,Y 249.427,Z 319.407,A -85,B 0,C 180,E1 -18729.733,E2 -18729.733} C_VEL
LIN {X 0,Y 249.208,Z 319.436,A -85,B 0,C 180,E1 -18734.703,E2 -18734.703} C_VEL
LIN {X 0,Y 249.142,Z 319.447,A -85,B 0,C 180,E1 -18738.077,E2 -18738.077} C_VEL
LIN {X 0,Y 249.087,Z 319.445,A -85,B 0,C 180,E1 -18741.518,E2 -18741.518} C_VEL
LIN {X 0,Y 249.119,Z 319.44,A -85,B 0,C 180,E1 -18745.475,E2 -18745.475} C_VEL
LIN {X 0,Y 249.086,Z 319.45,A -85,B 0,C 180,E1 -18748.993,E2 -18748.993} C_VEL
LIN {X 0,Y 249.033,Z 319.463,A -85,B 0,C 180,E1 -18752.425,E2 -18752.425} C_VEL
LIN {X 0,Y 249.05,Z 319.46,A -85,B 0,C 180,E1 -18756.342,E2 -18756.342} C_VEL
LIN {X 0,Y 249.008,Z 319.461,A -85,B 0,C 180,E1 -18760.478,E2 -18760.478} C_VEL
LIN {X 0,Y 248.988,Z 319.471,A -85,B 0,C 180,E1 -18764.883,E2 -18764.883} C_VEL
LIN {X 0,Y 249.045,Z 319.64,A -85,B 0,C 180,E1 -18765.521,E2 -18765.521} C_VEL
LIN {X 0,Y 251.115,Z 326.621,A -85,B 0,C 180,E1 -18769.083,E2 -18769.083} C_VEL
LIN {X 0,Y 253.208,Z 333.966,A -85,B 0,C 180,E1 -18772.467,E2 -18772.467} C_VEL
LIN {X 0,Y 255.631,Z 338.328,A -85,B 0,C 180,E1 -18773.131,E2 -18773.131} C_VEL
LIN {X 0,Y 263.335,Z 352.761,A -85,B 0,C 180,E1 -18775.137,E2 -18775.137} C_VEL
LIN {X 0,Y 270.344,Z 367.912,A -85,B 0,C 180,E1 -18776.872,E2 -18776.872} C_VEL
LIN {X 0,Y 273.65,Z 387.027,A -85,B 0,C 180,E1 -18778.037,E2 -18778.037} C_VEL
LIN {X 0,Y 273.955,Z 391.453,A -85,B 0,C 180,E1 -18778.229,E2 -18778.229} C_VEL
LIN {X 0,Y 271.645,Z 443.54,A -85,B 0,C 180,E1 -18779.605,E2 -18779.605} C_VEL
LIN {X 0,Y 270.347,Z 456.874,A -85,B 0,C 180,E1 -18780.219,E2 -18780.219} C_VEL
LIN {X 0,Y 268.507,Z 469.079,A -85,B 0,C 180,E1 -18781.037,E2 -18781.037} C_VEL
LIN {X 0,Y 266.36,Z 480.369,A -85,B 0,C 180,E1 -18782.073,E2 -18782.073} C_VEL
LIN {X 0,Y 263.671,Z 492.022,A -85,B 0,C 180,E1 -18783.482,E2 -18783.482} C_VEL
LIN {X 0,Y 260.957,Z 502.5,A -85,B 0,C 180,E1 -18785.114,E2 -18785.114} C_VEL
LIN {X 0,Y 258.371,Z 511.094,A -85,B 0,C 180,E1 -18786.77,E2 -18786.77} C_VEL
LIN {X 0,Y 255.892,Z 519.028,A -85,B 0,C 180,E1 -18788.659,E2 -18788.659} C_VEL
LIN {X 0,Y 253.442,Z 526.835,A -85,B 0,C 180,E1 -18790.983,E2 -18790.983} C_VEL
